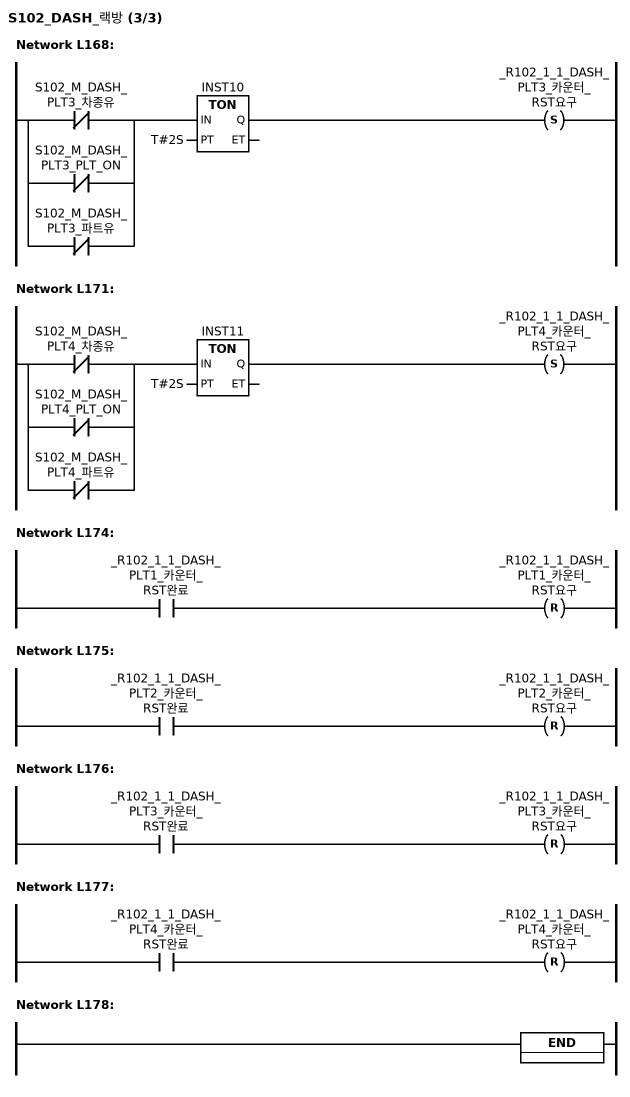
(* Rung L168 *)
INST10(IN := NOT S102_M_DASH_PLT3_차종유 OR NOT S102_M_DASH_PLT3_PLT_ON OR NOT S102_M_DASH_PLT3_파트유, PT := T#2S);
IF INST10.Q THEN _R102_1_1_DASH_PLT3_카운터_RST요구 := TRUE; END_IF;
(* Rung L171 *)
INST11(IN := NOT S102_M_DASH_PLT4_차종유 OR NOT S102_M_DASH_PLT4_PLT_ON OR NOT S102_M_DASH_PLT4_파트유, PT := T#2S);
IF INST11.Q THEN _R102_1_1_DASH_PLT4_카운터_RST요구 := TRUE; END_IF;
(* Rung L174 *)
IF _R102_1_1_DASH_PLT1_카운터_RST완료 THEN _R102_1_1_DASH_PLT1_카운터_RST요구 := FALSE; END_IF;
(* Rung L175 *)
IF _R102_1_1_DASH_PLT2_카운터_RST완료 THEN _R102_1_1_DASH_PLT2_카운터_RST요구 := FALSE; END_IF;
(* Rung L176 *)
IF _R102_1_1_DASH_PLT3_카운터_RST완료 THEN _R102_1_1_DASH_PLT3_카운터_RST요구 := FALSE; END_IF;
(* Rung L177 *)
IF _R102_1_1_DASH_PLT4_카운터_RST완료 THEN _R102_1_1_DASH_PLT4_카운터_RST요구 := FALSE; END_IF;
(* Rung L178 *)
END();
END_PROGRAM

PROGRAM S102_DASH_랙방_우선순위 (* task: 스캔 프로그램 *)
VAR_EXTERNAL
    S101_LH_M_APRON_PLT1_PLT_ON : BOOL; (* AT %MW1200.1 *)
    S101_LH_M_APRON_PLT1_로딩완료 : BOOL; (* AT %MW1200.10 *)
    S101_LH_M_APRON_PLT1_차종유 : BOOL; (* AT %MW1200.8 *)
    S101_LH_M_APRON_PLT1_파트유 : BOOL; (* AT %MW1200.3 *)
    S101_LH_M_APRON_PLT2_PLT_ON : BOOL; (* AT %MW1201.1 *)
    S101_LH_M_APRON_PLT2_로딩완료 : BOOL; (* AT %MW1201.10 *)
    S101_LH_M_APRON_PLT2_차종유 : BOOL; (* AT %MW1201.8 *)
    S101_LH_M_APRON_PLT2_파트유 : BOOL; (* AT %MW1201.3 *)
    S101_LH_M_APRON_PLT_PRIORITY1 : WORD; (* AT %MW1208 *)
    S101_LH_M_APRON_PLT_PRIORITY2 : WORD; (* AT %MW1209 *)
    S101_LH_M_APRON_PLT_PRIORITY3 : WORD; (* AT %MW1210 *)
    S101_LH_M_APRON_PLT_PRIORITY4 : WORD; (* AT %MW1211 *)
    S101_LH_M_APRON_PLT_PRIORITY5 : WORD; (* AT %MW1212 *)
    S101_LH_M_APRON_PLT_PRIORITY6 : WORD; (* AT %MW1213 *)
    S101_LH_M_APRON_PLT_PRIORITY7 : WORD; (* AT %MW1214 *)
    S101_LH_M_APRON_PLT_PRIORITY8 : WORD; (* AT %MW1215 *)
    S101_RH_M_APRON_PLT1_PLT_ON : BOOL; (* AT %MW1250.1 *)
    S101_RH_M_APRON_PLT1_로딩완료 : BOOL; (* AT %MW1250.10 *)
    S101_RH_M_APRON_PLT1_차종유 : BOOL; (* AT %MW1250.8 *)
    S101_RH_M_APRON_PLT1_파트유 : BOOL; (* AT %MW1250.3 *)
    S101_RH_M_APRON_PLT2_PLT_ON : BOOL; (* AT %MW1251.1 *)
    S101_RH_M_APRON_PLT2_로딩완료 : BOOL; (* AT %MW1251.10 *)
    S101_RH_M_APRON_PLT2_차종유 : BOOL; (* AT %MW1251.8 *)
    S101_RH_M_APRON_PLT2_파트유 : BOOL; (* AT %MW1251.3 *)
    S101_RH_M_APRON_PLT_PRIORITY1 : WORD; (* AT %MW1258 *)
    S101_RH_M_APRON_PLT_PRIORITY2 : WORD; (* AT %MW1259 *)
    S101_RH_M_APRON_PLT_PRIORITY3 : WORD; (* AT %MW1260 *)
    S101_RH_M_APRON_PLT_PRIORITY4 : WORD; (* AT %MW1261 *)
    S101_RH_M_APRON_PLT_PRIORITY5 : WORD; (* AT %MW1262 *)
    S101_RH_M_APRON_PLT_PRIORITY6 : WORD; (* AT %MW1263 *)
    S101_RH_M_APRON_PLT_PRIORITY7 : WORD; (* AT %MW1264 *)
    S101_RH_M_APRON_PLT_PRIORITY8 : WORD; (* AT %MW1265 *)
    S102_M_DASH_PLT1_PLT_ON : BOOL; (* AT %MW1700.1 *)
    S102_M_DASH_PLT1_로딩완료 : BOOL; (* AT %MW1700.10 *)
    S102_M_DASH_PLT1_차종유 : BOOL; (* AT %MW1700.8 *)
    S102_M_DASH_PLT1_파트유 : BOOL; (* AT %MW1700.3 *)
    S102_M_DASH_PLT2_PLT_ON : BOOL; (* AT %MW1701.1 *)
    S102_M_DASH_PLT2_로딩완료 : BOOL; (* AT %MW1701.10 *)
    S102_M_DASH_PLT2_차종유 : BOOL; (* AT %MW1701.8 *)
    S102_M_DASH_PLT2_파트유 : BOOL; (* AT %MW1701.3 *)
    S102_M_DASH_PLT3_PLT_ON : BOOL; (* AT %MW1702.1 *)
    S102_M_DASH_PLT3_로딩완료 : BOOL; (* AT %MW1702.10 *)
    S102_M_DASH_PLT3_차종유 : BOOL; (* AT %MW1702.8 *)
    S102_M_DASH_PLT3_파트유 : BOOL; (* AT %MW1702.3 *)
    S102_M_DASH_PLT4_PLT_ON : BOOL; (* AT %MW1703.1 *)
    S102_M_DASH_PLT4_로딩완료 : BOOL; (* AT %MW1703.10 *)
    S102_M_DASH_PLT4_차종유 : BOOL; (* AT %MW1703.8 *)
    S102_M_DASH_PLT4_파트유 : BOOL; (* AT %MW1703.3 *)
    S102_M_DASH_PLT_PRIORITY1 : WORD; (* AT %MW1708 *)
    S102_M_DASH_PLT_PRIORITY2 : WORD; (* AT %MW1709 *)
    S102_M_DASH_PLT_PRIORITY3 : WORD; (* AT %MW1710 *)
    S102_M_DASH_PLT_PRIORITY4 : WORD; (* AT %MW1711 *)
    S102_M_DASH_PLT_PRIORITY5 : WORD; (* AT %MW1712 *)
    S102_M_DASH_PLT_PRIORITY6 : WORD; (* AT %MW1713 *)
    S102_M_DASH_PLT_PRIORITY7 : WORD; (* AT %MW1714 *)
    S102_M_DASH_PLT_PRIORITY8 : WORD; (* AT %MW1715 *)
END_VAR
VAR
    _p1 : BOOL;
    _t2 : BOOL;
    _t3 : BOOL;
    _t4 : BOOL;
    _t5 : BOOL;
    _t6 : BOOL;
    _t7 : BOOL;
    _t8 : BOOL;
    _t9 : BOOL;
    _p10 : BOOL;
    _t11 : BOOL;
    _t12 : BOOL;
    _t13 : BOOL;
    _t14 : BOOL;
    _t15 : BOOL;
    _t16 : BOOL;
    _t17 : BOOL;
    _t18 : BOOL;
    _p19 : BOOL;
    _t20 : BOOL;
    _t21 : BOOL;
    _t22 : BOOL;
    _t23 : BOOL;
    _t24 : BOOL;
    _t25 : BOOL;
    _t26 : BOOL;
    _t27 : BOOL;
    _p28 : BOOL;
    _t29 : BOOL;
    _t30 : BOOL;
    _t31 : BOOL;
    _t32 : BOOL;
    _t33 : BOOL;
    _t34 : BOOL;
    _t35 : BOOL;
    _t36 : BOOL;
END_VAR
(* 랙방번호 우선순위버퍼 전송 *)
(* Rung L1: network not rendered *)
(* not connected or not rendered: S102_M_DASH_PLT1_로딩완료, S102_M_DASH_PLT1_PLT_ON, S102_M_DASH_PLT1_파트유, S102_M_DASH_PLT1_차종유, S102_M_DASH_PLT2_로딩완료, S102_M_DASH_PLT2_PLT_ON, S102_M_DASH_PLT2_파트유, S102_M_DASH_PLT2_차종유, S102_M_DASH_PLT3_로딩완료, S102_M_DASH_PLT3_PLT_ON, S102_M_DASH_PLT3_파트유, S102_M_DASH_PLT3_차종유, S102_M_DASH_PLT4_로딩완료, S102_M_DASH_PLT4_PLT_ON, S102_M_DASH_PLT4_파트유, S102_M_DASH_PLT4_차종유, S102_M_DASH_PLT_PRIORITY8, 0, S102_M_DASH_PLT_PRIORITY8, 2, S102_M_DASH_PLT_PRIORITY8, 3, S102_M_DASH_PLT_PRIORITY8, 4, S102_M_DASH_PLT_PRIORITY8 *)
(* 우선순위8->우선순위7 *)
(* Rung L15: network not rendered *)
(* not connected or not rendered: S102_M_DASH_PLT_PRIORITY8, 0, S102_M_DASH_PLT_PRIORITY7, 0, S102_M_DASH_PLT_PRIORITY8, S102_M_DASH_PLT_PRIORITY7, 0, S102_M_DASH_PLT_PRIORITY8 *)
(* 우선순위7->우선순위6 *)
(* Rung L24: network not rendered *)
(* not connected or not rendered: S102_M_DASH_PLT_PRIORITY7, 0, S102_M_DASH_PLT_PRIORITY6, 0, S102_M_DASH_PLT_PRIORITY7, S102_M_DASH_PLT_PRIORITY6, 0, S102_M_DASH_PLT_PRIORITY7 *)
(* 우선순위6->우선순위5 *)
(* Rung L33: network not rendered *)
(* not connected or not rendered: S102_M_DASH_PLT_PRIORITY6, 0, S102_M_DASH_PLT_PRIORITY5, 0, S102_M_DASH_PLT_PRIORITY6, S102_M_DASH_PLT_PRIORITY5, 0, S102_M_DASH_PLT_PRIORITY6 *)
(* 우선순위5->우선순위4 *)
(* Rung L42: network not rendered *)
(* not connected or not rendered: S102_M_DASH_PLT_PRIORITY5, 0, S102_M_DASH_PLT_PRIORITY4, 0, S102_M_DASH_PLT_PRIORITY5, S102_M_DASH_PLT_PRIORITY4, 0, S102_M_DASH_PLT_PRIORITY5 *)
(* 우선순위4->우선순위3 *)
(* Rung L51: network not rendered *)
(* not connected or not rendered: S102_M_DASH_PLT_PRIORITY4, 0, S102_M_DASH_PLT_PRIORITY3, 0, S102_M_DASH_PLT_PRIORITY4, S102_M_DASH_PLT_PRIORITY3, 0, S102_M_DASH_PLT_PRIORITY4 *)
(* 우선순위3->우선순위2 *)
(* Rung L60: network not rendered *)
(* not connected or not rendered: S102_M_DASH_PLT_PRIORITY3, S102_M_DASH_PLT_PRIORITY2, S102_M_DASH_PLT_PRIORITY3, S102_M_DASH_PLT_PRIORITY2, S102_M_DASH_PLT_PRIORITY3 *)
(* 우선순위2->우선순위1 *)
(* Rung L69: network not rendered *)
(* not connected or not rendered: S102_M_DASH_PLT_PRIORITY2, 0, S102_M_DASH_PLT_PRIORITY1, 0, S102_M_DASH_PLT_PRIORITY2, S102_M_DASH_PLT_PRIORITY1, 0, S102_M_DASH_PLT_PRIORITY2 *)

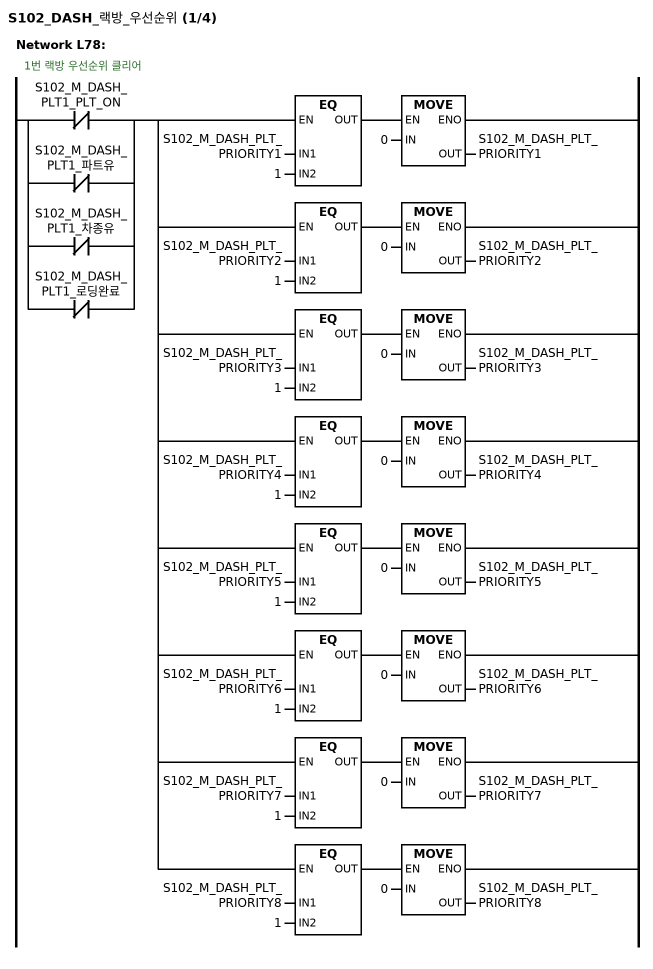
(* 1번 랙방 우선순위 클리어 *)
(* Rung L78 *)
_p1 := NOT S102_M_DASH_PLT1_PLT_ON OR NOT S102_M_DASH_PLT1_파트유 OR NOT S102_M_DASH_PLT1_차종유 OR NOT S102_M_DASH_PLT1_로딩완료;
IF _p1 THEN _t2 := S102_M_DASH_PLT_PRIORITY1 = 1; END_IF;
IF _t2 THEN S102_M_DASH_PLT_PRIORITY1 := 0; END_IF;
IF _p1 THEN _t3 := S102_M_DASH_PLT_PRIORITY2 = 1; END_IF;
IF _t3 THEN S102_M_DASH_PLT_PRIORITY2 := 0; END_IF;
IF _p1 THEN _t4 := S102_M_DASH_PLT_PRIORITY3 = 1; END_IF;
IF _t4 THEN S102_M_DASH_PLT_PRIORITY3 := 0; END_IF;
IF _p1 THEN _t5 := S102_M_DASH_PLT_PRIORITY4 = 1; END_IF;
IF _t5 THEN S102_M_DASH_PLT_PRIORITY4 := 0; END_IF;
IF _p1 THEN _t6 := S102_M_DASH_PLT_PRIORITY5 = 1; END_IF;
IF _t6 THEN S102_M_DASH_PLT_PRIORITY5 := 0; END_IF;
IF _p1 THEN _t7 := S102_M_DASH_PLT_PRIORITY6 = 1; END_IF;
IF _t7 THEN S102_M_DASH_PLT_PRIORITY6 := 0; END_IF;
IF _p1 THEN _t8 := S102_M_DASH_PLT_PRIORITY7 = 1; END_IF;
IF _t8 THEN S102_M_DASH_PLT_PRIORITY7 := 0; END_IF;
IF _p1 THEN _t9 := S102_M_DASH_PLT_PRIORITY8 = 1; END_IF;
IF _t9 THEN S102_M_DASH_PLT_PRIORITY8 := 0; END_IF;

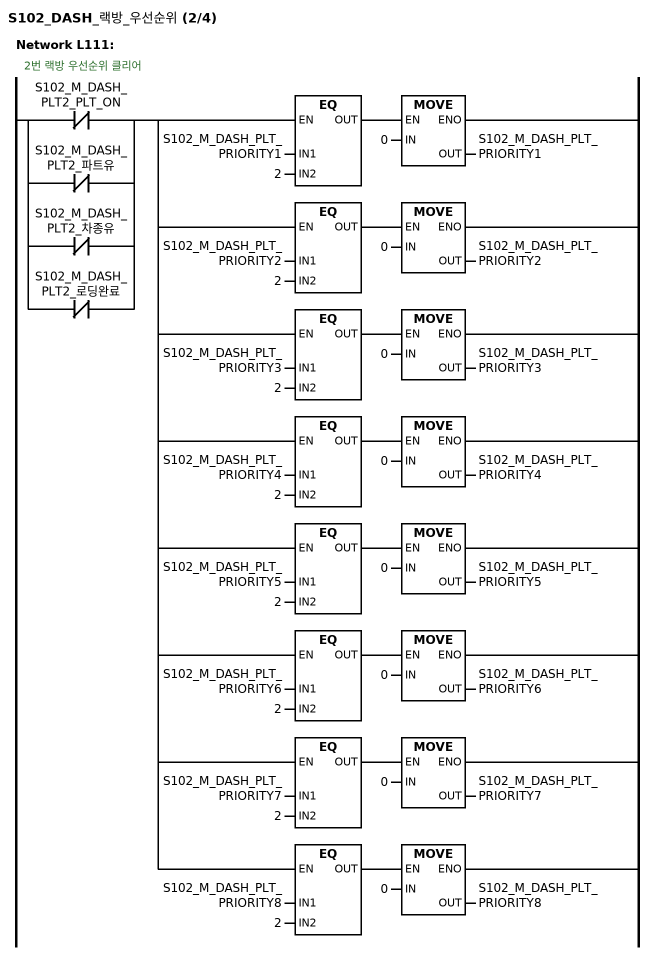
(* 2번 랙방 우선순위 클리어 *)
(* Rung L111 *)
_p10 := NOT S102_M_DASH_PLT2_PLT_ON OR NOT S102_M_DASH_PLT2_파트유 OR NOT S102_M_DASH_PLT2_차종유 OR NOT S102_M_DASH_PLT2_로딩완료;
IF _p10 THEN _t11 := S102_M_DASH_PLT_PRIORITY1 = 2; END_IF;
IF _t11 THEN S102_M_DASH_PLT_PRIORITY1 := 0; END_IF;
IF _p10 THEN _t12 := S102_M_DASH_PLT_PRIORITY2 = 2; END_IF;
IF _t12 THEN S102_M_DASH_PLT_PRIORITY2 := 0; END_IF;
IF _p10 THEN _t13 := S102_M_DASH_PLT_PRIORITY3 = 2; END_IF;
IF _t13 THEN S102_M_DASH_PLT_PRIORITY3 := 0; END_IF;
IF _p10 THEN _t14 := S102_M_DASH_PLT_PRIORITY4 = 2; END_IF;
IF _t14 THEN S102_M_DASH_PLT_PRIORITY4 := 0; END_IF;
IF _p10 THEN _t15 := S102_M_DASH_PLT_PRIORITY5 = 2; END_IF;
IF _t15 THEN S102_M_DASH_PLT_PRIORITY5 := 0; END_IF;
IF _p10 THEN _t16 := S102_M_DASH_PLT_PRIORITY6 = 2; END_IF;
IF _t16 THEN S102_M_DASH_PLT_PRIORITY6 := 0; END_IF;
IF _p10 THEN _t17 := S102_M_DASH_PLT_PRIORITY7 = 2; END_IF;
IF _t17 THEN S102_M_DASH_PLT_PRIORITY7 := 0; END_IF;
IF _p10 THEN _t18 := S102_M_DASH_PLT_PRIORITY8 = 2; END_IF;
IF _t18 THEN S102_M_DASH_PLT_PRIORITY8 := 0; END_IF;

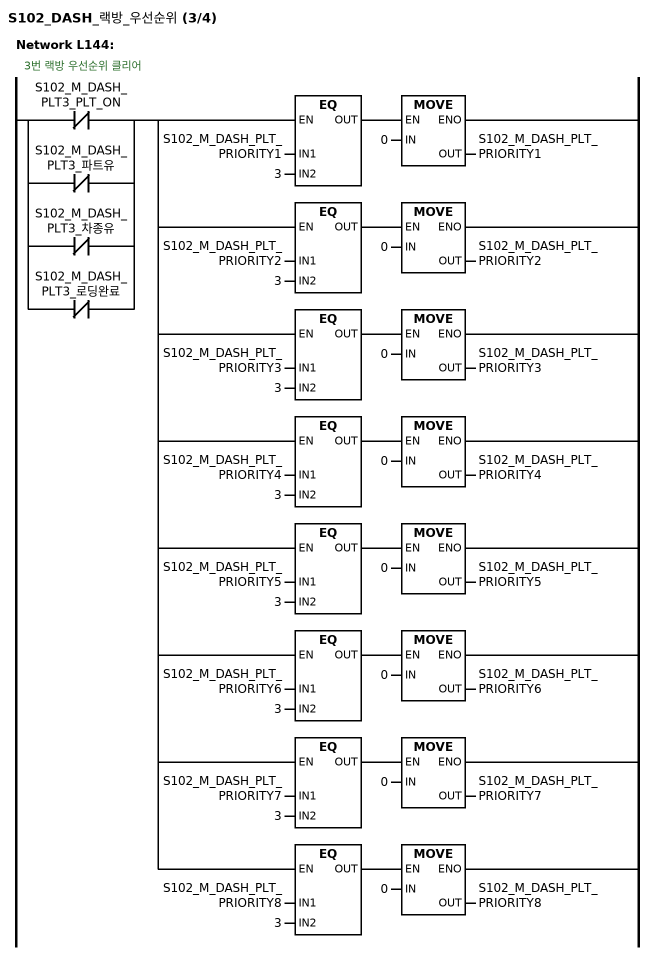
(* 3번 랙방 우선순위 클리어 *)
(* Rung L144 *)
_p19 := NOT S102_M_DASH_PLT3_PLT_ON OR NOT S102_M_DASH_PLT3_파트유 OR NOT S102_M_DASH_PLT3_차종유 OR NOT S102_M_DASH_PLT3_로딩완료;
IF _p19 THEN _t20 := S102_M_DASH_PLT_PRIORITY1 = 3; END_IF;
IF _t20 THEN S102_M_DASH_PLT_PRIORITY1 := 0; END_IF;
IF _p19 THEN _t21 := S102_M_DASH_PLT_PRIORITY2 = 3; END_IF;
IF _t21 THEN S102_M_DASH_PLT_PRIORITY2 := 0; END_IF;
IF _p19 THEN _t22 := S102_M_DASH_PLT_PRIORITY3 = 3; END_IF;
IF _t22 THEN S102_M_DASH_PLT_PRIORITY3 := 0; END_IF;
IF _p19 THEN _t23 := S102_M_DASH_PLT_PRIORITY4 = 3; END_IF;
IF _t23 THEN S102_M_DASH_PLT_PRIORITY4 := 0; END_IF;
IF _p19 THEN _t24 := S102_M_DASH_PLT_PRIORITY5 = 3; END_IF;
IF _t24 THEN S102_M_DASH_PLT_PRIORITY5 := 0; END_IF;
IF _p19 THEN _t25 := S102_M_DASH_PLT_PRIORITY6 = 3; END_IF;
IF _t25 THEN S102_M_DASH_PLT_PRIORITY6 := 0; END_IF;
IF _p19 THEN _t26 := S102_M_DASH_PLT_PRIORITY7 = 3; END_IF;
IF _t26 THEN S102_M_DASH_PLT_PRIORITY7 := 0; END_IF;
IF _p19 THEN _t27 := S102_M_DASH_PLT_PRIORITY8 = 3; END_IF;
IF _t27 THEN S102_M_DASH_PLT_PRIORITY8 := 0; END_IF;

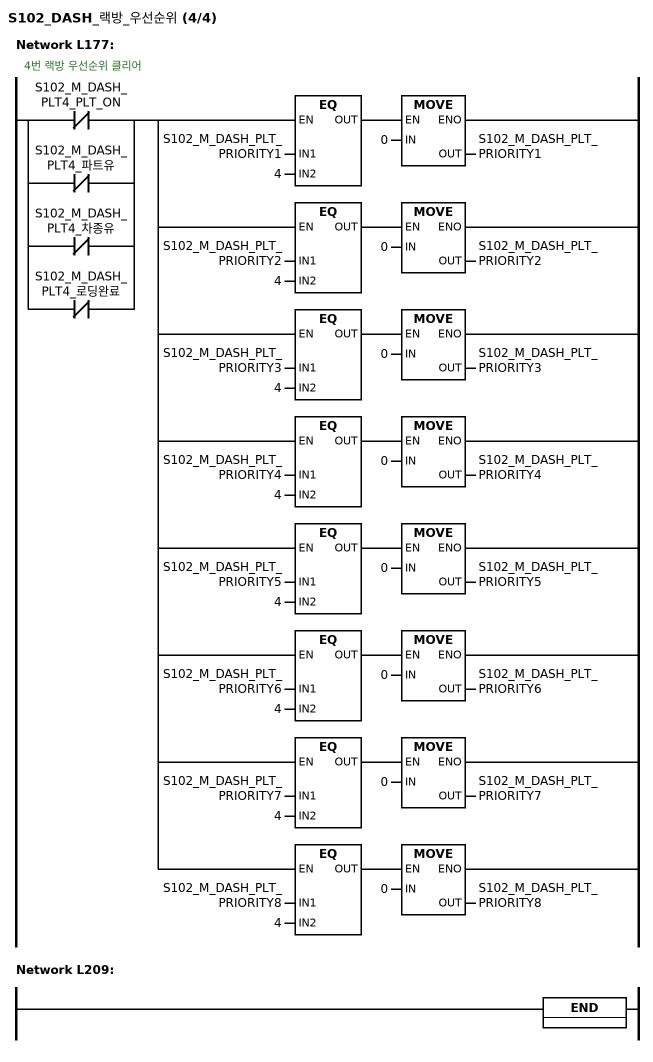
(* 4번 랙방 우선순위 클리어 *)
(* Rung L177 *)
_p28 := NOT S102_M_DASH_PLT4_PLT_ON OR NOT S102_M_DASH_PLT4_파트유 OR NOT S102_M_DASH_PLT4_차종유 OR NOT S102_M_DASH_PLT4_로딩완료;
IF _p28 THEN _t29 := S102_M_DASH_PLT_PRIORITY1 = 4; END_IF;
IF _t29 THEN S102_M_DASH_PLT_PRIORITY1 := 0; END_IF;
IF _p28 THEN _t30 := S102_M_DASH_PLT_PRIORITY2 = 4; END_IF;
IF _t30 THEN S102_M_DASH_PLT_PRIORITY2 := 0; END_IF;
IF _p28 THEN _t31 := S102_M_DASH_PLT_PRIORITY3 = 4; END_IF;
IF _t31 THEN S102_M_DASH_PLT_PRIORITY3 := 0; END_IF;
IF _p28 THEN _t32 := S102_M_DASH_PLT_PRIORITY4 = 4; END_IF;
IF _t32 THEN S102_M_DASH_PLT_PRIORITY4 := 0; END_IF;
IF _p28 THEN _t33 := S102_M_DASH_PLT_PRIORITY5 = 4; END_IF;
IF _t33 THEN S102_M_DASH_PLT_PRIORITY5 := 0; END_IF;
IF _p28 THEN _t34 := S102_M_DASH_PLT_PRIORITY6 = 4; END_IF;
IF _t34 THEN S102_M_DASH_PLT_PRIORITY6 := 0; END_IF;
IF _p28 THEN _t35 := S102_M_DASH_PLT_PRIORITY7 = 4; END_IF;
IF _t35 THEN S102_M_DASH_PLT_PRIORITY7 := 0; END_IF;
IF _p28 THEN _t36 := S102_M_DASH_PLT_PRIORITY8 = 4; END_IF;
IF _t36 THEN S102_M_DASH_PLT_PRIORITY8 := 0; END_IF;
(* Rung L209 *)
END();
END_PROGRAM

PROGRAM S102_로보트 (* task: 스캔 프로그램 *)
VAR_EXTERNAL
    AWAYS_OFF : BOOL; (* AT %MW3.0 *)
    AWAYS_ON : BOOL; (* AT %MW3.1 *)
    MCP_M_부저_정지 : BOOL; (* AT %MW350.5 *)
    MCP_M_비상정지 : BOOL; (* AT %MW350.7 *)
    MCP_PBL_운전준비_ON : BOOL; (* AT %MW87630.0 *) (* 입력 접점 00 *)
    R101_1_1_M_I_RB_간섭무_2 : BOOL; (* AT %MW20042.1 *)
    R101_1_M_I_RB_간섭무_2 : BOOL; (* AT %MW20072.1 *)
    R101_2_M_I_RB_간섭무_2 : BOOL; (* AT %MW20062.1 *)
    R101_3_M_I_RB_간섭무_2 : BOOL; (* AT %MW20052.1 *)
    R102_1_1_I_RB_INPUT : ARRAY[0..3] OF WORD; (* AT %MW84090 *)
    R102_1_1_M_I_RB_1차_작업완료 : BOOL; (* AT %MW20091.2 *)
    R102_1_1_M_I_RB_2차_작업완료 : BOOL; (* AT %MW20091.3 *)
    R102_1_1_M_I_RB_3차_작업완료 : BOOL; (* AT %MW20091.4 *)
    R102_1_1_M_I_RB_4차_작업완료 : BOOL; (* AT %MW20091.5 *)
    R102_1_1_M_I_RB_5차_작업완료 : BOOL; (* AT %MW20091.6 *)
    R102_1_1_M_I_RB_6차_작업완료 : BOOL; (* AT %MW20091.7 *)
    R102_1_1_M_I_RB_7차_작업완료 : BOOL; (* AT %MW20091.8 *)
    R102_1_1_M_I_RB_PAUSE_보조 : BOOL; (* AT %MW20090.5 *)
    R102_1_1_M_I_RB_PLC_RUN_CHK_이상 : BOOL; (* AT %MW20090.7 *)
    R102_1_1_M_I_RB_간섭무_1 : BOOL; (* AT %MW20092.0 *)
    R102_1_1_M_I_RB_간섭무_10 : BOOL; (* AT %MW20092.9 *)
    R102_1_1_M_I_RB_간섭무_11 : BOOL; (* AT %MW20092.10 *)
    R102_1_1_M_I_RB_간섭무_12 : BOOL; (* AT %MW20092.11 *)
    R102_1_1_M_I_RB_간섭무_2 : BOOL; (* AT %MW20092.1 *)
    R102_1_1_M_I_RB_간섭무_3 : BOOL; (* AT %MW20092.2 *)
    R102_1_1_M_I_RB_간섭무_4 : BOOL; (* AT %MW20092.3 *)
    R102_1_1_M_I_RB_간섭무_5 : BOOL; (* AT %MW20092.4 *)
    R102_1_1_M_I_RB_간섭무_6 : BOOL; (* AT %MW20092.5 *)
    R102_1_1_M_I_RB_간섭무_7 : BOOL; (* AT %MW20092.6 *)
    R102_1_1_M_I_RB_간섭무_8 : BOOL; (* AT %MW20092.7 *)
    R102_1_1_M_I_RB_간섭무_9 : BOOL; (* AT %MW20092.8 *)
    R102_1_1_M_I_RB_비상정지 : BOOL; (* AT %MW20090.4 *)
    R102_1_1_M_I_RB_운전준비 : BOOL; (* AT %MW20090.0 *)
    R102_1_1_M_I_RB_원위치 : BOOL; (* AT %MW20090.3 *)
    R102_1_1_M_I_RB_이상 : BOOL; (* AT %MW20090.2 *)
    R102_1_1_M_I_RB_자동 : BOOL; (* AT %MW20090.1 *)
    R102_1_1_M_I_RB_최종작업완료 : BOOL; (* AT %MW20091.0 *)
    R102_1_1_M_I_RB_프로그램_이상 : BOOL; (* AT %MW20090.6 *)
    R102_1_1_M_O_RB_1_CYCLE_SET : BOOL; (* AT %MW21090.3 *)
    R102_1_1_M_O_RB_1차_작업완료_리셋 : BOOL; (* AT %MW21092.0 *)
    R102_1_1_M_O_RB_2차_작업완료_리셋 : BOOL; (* AT %MW21092.1 *)
    R102_1_1_M_O_RB_2차_진입OK : BOOL; (* AT %MW21091.8 *)
    R102_1_1_M_O_RB_3차_작업완료_리셋 : BOOL; (* AT %MW21092.2 *)
    R102_1_1_M_O_RB_3차_진입OK : BOOL; (* AT %MW21091.9 *)
    R102_1_1_M_O_RB_4차_작업완료_리셋 : BOOL; (* AT %MW21092.3 *)
    R102_1_1_M_O_RB_4차_진입OK : BOOL; (* AT %MW21091.10 *)
    R102_1_1_M_O_RB_5차_작업완료_리셋 : BOOL; (* AT %MW21092.4 *)
    R102_1_1_M_O_RB_5차_진입OK : BOOL; (* AT %MW21091.11 *)
    R102_1_1_M_O_RB_6차_작업완료_리셋 : BOOL; (* AT %MW21092.5 *)
    R102_1_1_M_O_RB_6차_진입OK : BOOL; (* AT %MW21091.12 *)
    R102_1_1_M_O_RB_7차_작업완료_리셋 : BOOL; (* AT %MW21092.6 *)
    R102_1_1_M_O_RB_7차_진입OK : BOOL; (* AT %MW21091.13 *)
    R102_1_1_M_O_RB_ATD_OK : BOOL; (* AT %MW21090.6 *)
    R102_1_1_M_O_RB_PLT_10_진입OK : BOOL; (* AT %MW21093.10 *)
    R102_1_1_M_O_RB_PLT_11_진입OK : BOOL; (* AT %MW21093.11 *)
    R102_1_1_M_O_RB_PLT_12_진입OK : BOOL; (* AT %MW21093.12 *)
    R102_1_1_M_O_RB_PLT_1_진입OK : BOOL; (* AT %MW21093.1 *)
    R102_1_1_M_O_RB_PLT_2_진입OK : BOOL; (* AT %MW21093.2 *)
    R102_1_1_M_O_RB_PLT_3_진입OK : BOOL; (* AT %MW21093.3 *)
    R102_1_1_M_O_RB_PLT_4_진입OK : BOOL; (* AT %MW21093.4 *)
    R102_1_1_M_O_RB_PLT_5_진입OK : BOOL; (* AT %MW21093.5 *)
    R102_1_1_M_O_RB_PLT_6_진입OK : BOOL; (* AT %MW21093.6 *)
    R102_1_1_M_O_RB_PLT_7_진입OK : BOOL; (* AT %MW21093.7 *)
    R102_1_1_M_O_RB_PLT_8_진입OK : BOOL; (* AT %MW21093.8 *)
    R102_1_1_M_O_RB_PLT_9_진입OK : BOOL; (* AT %MW21093.9 *)
    R102_1_1_M_O_RB_PLT_카운터리셋_보조 : BOOL; (* AT %MW21090.10 *)
    R102_1_1_M_O_RB_RESTART_OK : BOOL; (* AT %MW21090.2 *)
    R102_1_1_M_O_RB_START_OK : BOOL; (* AT %MW21090.0 *)
    R102_1_1_M_O_RB_TEST_MODE_5000회 : BOOL; (* AT %MW21090.12 *)
    R102_1_1_M_O_RB_TIP_교체_시작 : BOOL; (* AT %MW21090.7 *)
    R102_1_1_M_O_RB_TIP_교체_완료 : BOOL; (* AT %MW21090.8 *)
    R102_1_1_M_O_RB_VIP_MODE : BOOL; (* AT %MW21090.11 *)
    R102_1_1_M_O_RB_냉각수_차단_요청 : BOOL; (* AT %MW21090.9 *)
    R102_1_1_M_O_RB_진입OK_AX차종 : BOOL; (* AT %MW21091.0 *)
    R102_1_1_M_O_RB_진입OK_B차종 : BOOL; (* AT %MW21091.1 *)
    R102_1_1_M_O_RB_진입OK_C차종 : BOOL; (* AT %MW21091.2 *)
    R102_1_1_M_O_RB_진입OK_D차종 : BOOL; (* AT %MW21091.3 *)
    R102_1_1_M_O_RB_진입OK_E차종 : BOOL; (* AT %MW21091.4 *)
    R102_1_1_M_O_RB_진입OK_F차종 : BOOL; (* AT %MW21091.5 *)
    R102_1_1_M_O_RB_진입OK_G차종 : BOOL; (* AT %MW21091.6 *)
    R102_1_1_M_O_RB_진입OK_H차종 : BOOL; (* AT %MW21091.7 *)
    R102_1_1_M_O_RB_최종_작업완료_리셋 : BOOL; (* AT %MW21090.5 *)
    R102_1_1_M_O_RB_프로그램_OK : BOOL; (* AT %MW21090.1 *)
    R102_1_1_M_RB_PROG_NO : WORD; (* AT %MW20094 *)
    R102_1_1_M_STN_차종_NONE : BOOL; (* AT %MW1502.3 *)
    R102_1_1_M_STN_차종_ON : BOOL; (* AT %MW1502.2 *)
    R102_1_1_M_차종1_AX : BOOL; (* AT %MW10041.0 *) (* R102_1_1_M_차종1_AX *)
    R102_1_1_O_RB_OUTPUT : ARRAY[0..3] OF WORD; (* AT %MW94090 *)
    R102_1_I_RB_INPUT : ARRAY[0..3] OF WORD; (* AT %MW84080 *)
    R102_1_M_I_RB_1차_작업완료 : BOOL; (* AT %MW20081.2 *)
    R102_1_M_I_RB_2차_작업완료 : BOOL; (* AT %MW20081.3 *)
    R102_1_M_I_RB_3차_작업완료 : BOOL; (* AT %MW20081.4 *)
    R102_1_M_I_RB_4차_작업완료 : BOOL; (* AT %MW20081.5 *)
    R102_1_M_I_RB_5차_작업완료 : BOOL; (* AT %MW20081.6 *)
    R102_1_M_I_RB_6차_작업완료 : BOOL; (* AT %MW20081.7 *)
    R102_1_M_I_RB_7차_작업완료 : BOOL; (* AT %MW20081.8 *)
    R102_1_M_I_RB_PAUSE_보조 : BOOL; (* AT %MW20080.5 *)
    R102_1_M_I_RB_PLC_RUN_CHK_이상 : BOOL; (* AT %MW20080.7 *)
    R102_1_M_I_RB_간섭무_1 : BOOL; (* AT %MW20082.0 *)
    R102_1_M_I_RB_간섭무_10 : BOOL; (* AT %MW20082.9 *)
    R102_1_M_I_RB_간섭무_11 : BOOL; (* AT %MW20082.10 *)
    R102_1_M_I_RB_간섭무_12 : BOOL; (* AT %MW20082.11 *)
    R102_1_M_I_RB_간섭무_2 : BOOL; (* AT %MW20082.1 *)
    R102_1_M_I_RB_간섭무_3 : BOOL; (* AT %MW20082.2 *)
    R102_1_M_I_RB_간섭무_4 : BOOL; (* AT %MW20082.3 *)
    R102_1_M_I_RB_간섭무_5 : BOOL; (* AT %MW20082.4 *)
    R102_1_M_I_RB_간섭무_6 : BOOL; (* AT %MW20082.5 *)
    R102_1_M_I_RB_간섭무_7 : BOOL; (* AT %MW20082.6 *)
    R102_1_M_I_RB_간섭무_8 : BOOL; (* AT %MW20082.7 *)
    R102_1_M_I_RB_간섭무_9 : BOOL; (* AT %MW20082.8 *)
    R102_1_M_I_RB_비상정지 : BOOL; (* AT %MW20080.4 *)
    R102_1_M_I_RB_운전준비 : BOOL; (* AT %MW20080.0 *)
    R102_1_M_I_RB_원위치 : BOOL; (* AT %MW20080.3 *)
    R102_1_M_I_RB_이상 : BOOL; (* AT %MW20080.2 *)
    R102_1_M_I_RB_자동 : BOOL; (* AT %MW20080.1 *)
    R102_1_M_I_RB_최종작업완료 : BOOL; (* AT %MW20081.0 *)
    R102_1_M_I_RB_프로그램_이상 : BOOL; (* AT %MW20080.6 *)
    R102_1_M_O_RB_1_CYCLE_SET : BOOL; (* AT %MW21080.3 *)
    R102_1_M_O_RB_1차_작업완료_리셋 : BOOL; (* AT %MW21082.0 *)
    R102_1_M_O_RB_2차_작업완료_리셋 : BOOL; (* AT %MW21082.1 *)
    R102_1_M_O_RB_2차_진입OK : BOOL; (* AT %MW21081.8 *)
    R102_1_M_O_RB_3차_작업완료_리셋 : BOOL; (* AT %MW21082.2 *)
    R102_1_M_O_RB_3차_진입OK : BOOL; (* AT %MW21081.9 *)
    R102_1_M_O_RB_4차_작업완료_리셋 : BOOL; (* AT %MW21082.3 *)
    R102_1_M_O_RB_4차_진입OK : BOOL; (* AT %MW21081.10 *)
    R102_1_M_O_RB_5차_작업완료_리셋 : BOOL; (* AT %MW21082.4 *)
    R102_1_M_O_RB_5차_진입OK : BOOL; (* AT %MW21081.11 *)
    R102_1_M_O_RB_6차_작업완료_리셋 : BOOL; (* AT %MW21082.5 *)
    R102_1_M_O_RB_6차_진입OK : BOOL; (* AT %MW21081.12 *)
    R102_1_M_O_RB_7차_작업완료_리셋 : BOOL; (* AT %MW21082.6 *)
    R102_1_M_O_RB_7차_진입OK : BOOL; (* AT %MW21081.13 *)
    R102_1_M_O_RB_ATD_OK : BOOL; (* AT %MW21080.6 *)
    R102_1_M_O_RB_PLT_10_진입OK : BOOL; (* AT %MW21083.10 *)
    R102_1_M_O_RB_PLT_11_진입OK : BOOL; (* AT %MW21083.11 *)
    R102_1_M_O_RB_PLT_12_진입OK : BOOL; (* AT %MW21083.12 *)
    R102_1_M_O_RB_PLT_1_진입OK : BOOL; (* AT %MW21083.1 *)
    R102_1_M_O_RB_PLT_2_진입OK : BOOL; (* AT %MW21083.2 *)
    R102_1_M_O_RB_PLT_3_진입OK : BOOL; (* AT %MW21083.3 *)
    R102_1_M_O_RB_PLT_4_진입OK : BOOL; (* AT %MW21083.4 *)
    R102_1_M_O_RB_PLT_5_진입OK : BOOL; (* AT %MW21083.5 *)
    R102_1_M_O_RB_PLT_6_진입OK : BOOL; (* AT %MW21083.6 *)
    R102_1_M_O_RB_PLT_7_진입OK : BOOL; (* AT %MW21083.7 *)
    R102_1_M_O_RB_PLT_8_진입OK : BOOL; (* AT %MW21083.8 *)
    R102_1_M_O_RB_PLT_9_진입OK : BOOL; (* AT %MW21083.9 *)
    R102_1_M_O_RB_PLT_카운터리셋_보조 : BOOL; (* AT %MW21080.10 *)
    R102_1_M_O_RB_RESTART_OK : BOOL; (* AT %MW21080.2 *)
    R102_1_M_O_RB_START_OK : BOOL; (* AT %MW21080.0 *)
    R102_1_M_O_RB_TEST_MODE_5000회 : BOOL; (* AT %MW21080.12 *)
    R102_1_M_O_RB_TIP_교체_시작 : BOOL; (* AT %MW21080.7 *)
    R102_1_M_O_RB_TIP_교체_완료 : BOOL; (* AT %MW21080.8 *)
    R102_1_M_O_RB_VIP_MODE : BOOL; (* AT %MW21080.11 *)
    R102_1_M_O_RB_냉각수_차단_요청 : BOOL; (* AT %MW21080.9 *)
    R102_1_M_O_RB_진입OK_AX차종 : BOOL; (* AT %MW21081.0 *)
    R102_1_M_O_RB_진입OK_B차종 : BOOL; (* AT %MW21081.1 *)
    R102_1_M_O_RB_진입OK_C차종 : BOOL; (* AT %MW21081.2 *)
    R102_1_M_O_RB_진입OK_D차종 : BOOL; (* AT %MW21081.3 *)
    R102_1_M_O_RB_진입OK_E차종 : BOOL; (* AT %MW21081.4 *)
    R102_1_M_O_RB_진입OK_F차종 : BOOL; (* AT %MW21081.5 *)
    R102_1_M_O_RB_진입OK_G차종 : BOOL; (* AT %MW21081.6 *)
    R102_1_M_O_RB_진입OK_H차종 : BOOL; (* AT %MW21081.7 *)
    R102_1_M_O_RB_최종_작업완료_리셋 : BOOL; (* AT %MW21080.5 *)
    R102_1_M_O_RB_프로그램_OK : BOOL; (* AT %MW21080.1 *)
    R102_1_M_RB_PROG_NO : WORD; (* AT %MW20084 *)
    R102_1_M_STN_차종_ON : BOOL; (* AT %MW1502.4 *)
    R102_1_M_차종1_AX : BOOL; (* AT %MW10081.0 *) (* R102_1_M_차종1_AX *)
    R102_1_O_RB_OUTPUT : ARRAY[0..3] OF WORD; (* AT %MW94080 *)
    R103_1_M_I_RB_간섭무_2 : BOOL; (* AT %MW20102.1 *)
    S101_M_STN_DASH_로딩완료 : BOOL; (* AT %MW1001.12 *)
    S101_M_STN_LH_로딩완료 : BOOL; (* AT %MW1001.10 *)
    S101_M_STN_RH_로딩완료 : BOOL; (* AT %MW1001.11 *)
    S101_M_STN_차종_ON : BOOL; (* AT %MW1002.0 *)
    S101_M_공정_APRON_제품감지_ON : BOOL; (* AT %MW1001.3 *)
    S101_M_공정_DASH_제품감지_OFF : BOOL; (* AT %MW1001.6 *)
    S101_M_공정_DASH_제품감지_ON : BOOL; (* AT %MW1001.5 *)
    S101_M_공정_간섭무 : BOOL; (* AT %MW1004.1 *)
    S101_M_자동_운전중 : BOOL; (* AT %MW1000.4 *)
    S101_M_작업_완료 : BOOL; (* AT %MW1001.0 *)
    S101_M_차종1_AX : BOOL; (* AT %MW10021.0 *) (* S101_M_차종1_AX *)
    S102_M_DASH_PLT1_FAULT : BOOL; (* AT %MW1700.6 *)
    S102_M_DASH_PLT1_MATCH_OK : BOOL; (* AT %MW1700.5 *)
    S102_M_DASH_PLT1_PROG_OK : BOOL; (* AT %MW1700.0 *)
    S102_M_DASH_PLT1_차종코드 : WORD; (* AT %MW1716 *)
    S102_M_DASH_PLT2_FAULT : BOOL; (* AT %MW1701.6 *)
    S102_M_DASH_PLT2_MATCH_OK : BOOL; (* AT %MW1701.5 *)
    S102_M_DASH_PLT2_PROG_OK : BOOL; (* AT %MW1701.0 *)
    S102_M_DASH_PLT2_차종코드 : WORD; (* AT %MW1717 *)
    S102_M_DASH_PLT3_FAULT : BOOL; (* AT %MW1702.6 *)
    S102_M_DASH_PLT3_MATCH_OK : BOOL; (* AT %MW1702.5 *)
    S102_M_DASH_PLT3_PROG_OK : BOOL; (* AT %MW1702.0 *)
    S102_M_DASH_PLT3_차종코드 : WORD; (* AT %MW1718 *)
    S102_M_DASH_PLT4_FAULT : BOOL; (* AT %MW1703.6 *)
    S102_M_DASH_PLT4_MATCH_OK : BOOL; (* AT %MW1703.5 *)
    S102_M_DASH_PLT4_PROG_OK : BOOL; (* AT %MW1703.0 *)
    S102_M_DASH_PLT4_차종코드 : WORD; (* AT %MW1719 *)
    S102_M_DASH_PLT_PRIORITY1 : WORD; (* AT %MW1708 *)
    S102_M_STN_차종_NONE : BOOL; (* AT %MW1502.1 *)
    S102_M_STN_차종_ON : BOOL; (* AT %MW1502.0 *)
    S102_M_공정_간섭무 : BOOL; (* AT %MW1504.1 *)
    S102_M_공정_사양감지_OK : BOOL; (* AT %MW1501.5 *)
    S102_M_공정_제품감지_OFF : BOOL; (* AT %MW1501.4 *)
    S102_M_공정_제품감지_ON : BOOL; (* AT %MW1501.3 *)
    S102_M_자동_START : BOOL; (* AT %MW1500.5 *)
    S102_M_자동_운전중 : BOOL; (* AT %MW1500.4 *)
    S102_M_작업_완료 : BOOL; (* AT %MW1501.0 *)
    S102_M_차종1_AX : BOOL; (* AT %MW10061.0 *) (* S102_M_차종1_AX *)
    S102_M_총괄_이상 : BOOL; (* AT %MW1509.0 *)
    S103_M_FRT_안착OK_POS : BOOL; (* AT %MW2004.8 *)
    S103_M_STN_차종_NONE : BOOL; (* AT %MW2002.1 *)
    S103_M_STN_차종_ON : BOOL; (* AT %MW2002.0 *)
    S103_M_공정_제품감지_OFF : BOOL; (* AT %MW2001.4 *)
    S103_M_자동_운전중 : BOOL; (* AT %MW2000.4 *)
    S103_M_작업_완료 : BOOL; (* AT %MW2001.0 *)
    로보트제외 : BOOL;
    전체_M_GATE_CYCLE_정지 : BOOL; (* AT %MW308.0 *) (* 전체 M GATE CYCLE STOP *)
    전체_M_GATE_비상정지_정상 : BOOL; (* AT %MW308.4 *)
    전체_M_운전준비_보조 : BOOL; (* AT %MW308.5 *)
    전체_M_이상_리셋 : BOOL; (* AT %MW308.2 *) (* 전체 M 이상 리셋 *)
    전체_공정_M_총괄_비상정지_정상 : BOOL; (* AT %MW304.1 *) (* 전체 공정 M 총괄 비상정지 정상 *)
END_VAR
VAR
    INST1 : FB494_Robot_Hyundai_HMMI_v1;
    INST2 : FB494_Robot_Hyundai_HMMI_v1;
    _R102_1_1_PLT_언로딩완료 : BOOL;
END_VAR
(* ladder body could not be read *)
END_PROGRAM

PROGRAM S102_이상 (* task: 스캔 프로그램 *)
VAR
    INST10 : TON;
    INST11 : TON;
    INST12 : TON;
    INST13 : TON;
    INST14 : TON;
    INST15 : TON;
    INST16 : TON;
    INST17 : TON;
    INST18 : TON;
    INST19 : TON;
    INST20 : TON;
    INST21 : TON;
    INST22 : TON;
    INST23 : TON;
    INST24 : TON;
    INST25 : TON;
    INST26 : TON;
    INST27 : TON;
    INST28 : TON;
    INST8 : TON;
    INST9 : TON;
END_VAR
VAR_EXTERNAL
    R102_1_1_M_RB_통신이상 : BOOL; (* AT %MW1524.3 *)
    R102_1_1_M_차종3_LHD : BOOL; (* AT %MW10041.14 *) (* R102_1_1_M_차종3_LHD *)
    R102_1_1_M_차종3_RHD : BOOL; (* AT %MW10041.15 *) (* R102_1_1_M_차종3_RHD *)
    R102_1_1_M_차종5_AT : BOOL; (* AT %MW10043.1 *) (* R102_1_1_M_차종5_AT *)
    R102_1_1_M_차종5_MT : BOOL; (* AT %MW10043.0 *) (* R102_1_1_M_차종5_MT *)
    R102_1_M_RB_통신이상 : BOOL; (* AT %MW1524.4 *)
    S101_M_총괄_비상정지_이상 : BOOL; (* AT %MW1009.1 *)
    S102_6_20_PLC_BOX_CP_TRIP : BOOL; (* AT %MW86202.15 *) (* 입력 접점 15 *)
    S102_M_DASH_랙방1_2_통신이상 : BOOL; (* AT %MW1524.1 *)
    S102_M_DASH_랙방3_4_통신이상 : BOOL; (* AT %MW1524.2 *)
    S102_M_STN_DASH_로딩완료 : BOOL; (* AT %MW1501.8 *)
    S102_M_공정_간섭무 : BOOL; (* AT %MW1504.1 *)
    S102_M_공정_제품감지_ON : BOOL; (* AT %MW1501.3 *)
    S102_M_공정_통신이상 : BOOL; (* AT %MW1524.0 *)
    S102_M_사양_이상 : BOOL; (* AT %MW1516.0 *)
    S102_M_제품감지_이상 : BOOL; (* AT %MW1514.0 *)
    S102_M_차종1_AX : BOOL; (* AT %MW10061.0 *) (* S102_M_차종1_AX *)
    S102_M_총괄_CP_이상 : BOOL; (* AT %MW1509.7 *)
    S102_M_총괄_CT_이상 : BOOL; (* AT %MW1510.4 *)
    S102_M_총괄_EOCR_이상 : BOOL; (* AT %MW1509.8 *)
    S102_M_총괄_INV_이상 : BOOL; (* AT %MW1509.9 *)
    S102_M_총괄_LS_이상 : BOOL; (* AT %MW1509.15 *)
    S102_M_총괄_MATCH_이상 : BOOL; (* AT %MW1510.0 *)
    S102_M_총괄_MC_이상 : BOOL; (* AT %MW1509.13 *)
    S102_M_총괄_NFB_이상 : BOOL; (* AT %MW1509.11 *)
    S102_M_총괄_ROBOT_이상 : BOOL; (* AT %MW1510.1 *)
    S102_M_총괄_SAFETY_이상 : BOOL; (* AT %MW1509.2 *)
    S102_M_총괄_공기압_이상 : BOOL; (* AT %MW1509.3 *)
    S102_M_총괄_비상정지_이상 : BOOL; (* AT %MW1509.1 *)
    S102_M_총괄_사양_이상 : BOOL; (* AT %MW1509.6 *)
    S102_M_총괄_오버런_이상 : BOOL; (* AT %MW1509.12 *)
    S102_M_총괄_용점타점수_이상 : BOOL; (* AT %MW1510.2 *)
    S102_M_총괄_이상 : BOOL; (* AT %MW1509.0 *)
    S102_M_총괄_제품감지_이상 : BOOL; (* AT %MW1509.4 *)
    S102_M_총괄_차종_이상 : BOOL; (* AT %MW1509.5 *)
    S102_M_총괄_통신_이상 : BOOL; (* AT %MW1509.14 *)
    S102_PRS_I_AT_감지 : BOOL; (* AT %MW86201.8 *)
    S102_PRS_I_AX_파트_ON : BOOL; (* AT %MW86200.1 *)
    S102_PRS_I_LHD_감지 : BOOL; (* AT %MW86201.0 *)
    S102_PRS_I_MT_감지 : BOOL; (* AT %MW86201.9 *)
    S102_PRS_I_RHD_감지 : BOOL; (* AT %MW86201.1 *)
    S102_PRS_I_공용_파트_ON : BOOL; (* AT %MW86200.0 *)
    _0004_EB08_CFG_ER : BOOL; (* AT %MX59560 *) (* EB 구성 에러 *)
    _0004_EB08_DEER : BOOL; (* AT %MX59561 *) (* EB 운전 중 탈락 *)
    _0004_EB09_CFG_ER : BOOL; (* AT %MX59600 *) (* EB 구성 에러 *)
    _0004_EB09_DEER : BOOL; (* AT %MX59601 *) (* EB 운전 중 탈락 *)
    _0006_EB10_CFG_ER : BOOL; (* AT %MW186022.0 *) (* EB 구성 에러 *)
    _0006_EB10_DEER : BOOL; (* AT %MW186022.1 *) (* EB 운전 중 탈락 *)
    _0006_EB10_IO_DEER : BOOL; (* AT %MW186023.2 *) (* EB IO 탈락 에러 *)
    _0006_EB10_IO_TYER : BOOL; (* AT %MW186023.1 *) (* EB IO 타입 에러 *)
    _0006_EB20_CFG_ER : BOOL; (* AT %MW186028.0 *) (* EB 구성 에러 *)
    _0006_EB20_DEER : BOOL; (* AT %MW186028.1 *) (* EB 운전 중 탈락 *)
    _0006_EB20_IO_DEER : BOOL; (* AT %MW186029.2 *) (* EB IO 탈락 에러 *)
    _0006_EB20_IO_TYER : BOOL; (* AT %MW186029.1 *) (* EB IO 타입 에러 *)
    _0007_EB30_CFG_ER : BOOL; (* AT %MW187034.0 *) (* EB 구성 에러 *)
    _0007_EB30_DEER : BOOL; (* AT %MW187034.1 *) (* EB 운전 중 탈락 *)
    _0007_EB30_IO_DEER : BOOL; (* AT %MW187035.2 *) (* EB IO 탈락 에러 *)
    _0007_EB30_IO_TYER : BOOL; (* AT %MW187035.1 *) (* EB IO 타입 에러 *)
    전체_M_이상_리셋 : BOOL; (* AT %MW308.2 *) (* 전체 M 이상 리셋 *)
END_VAR

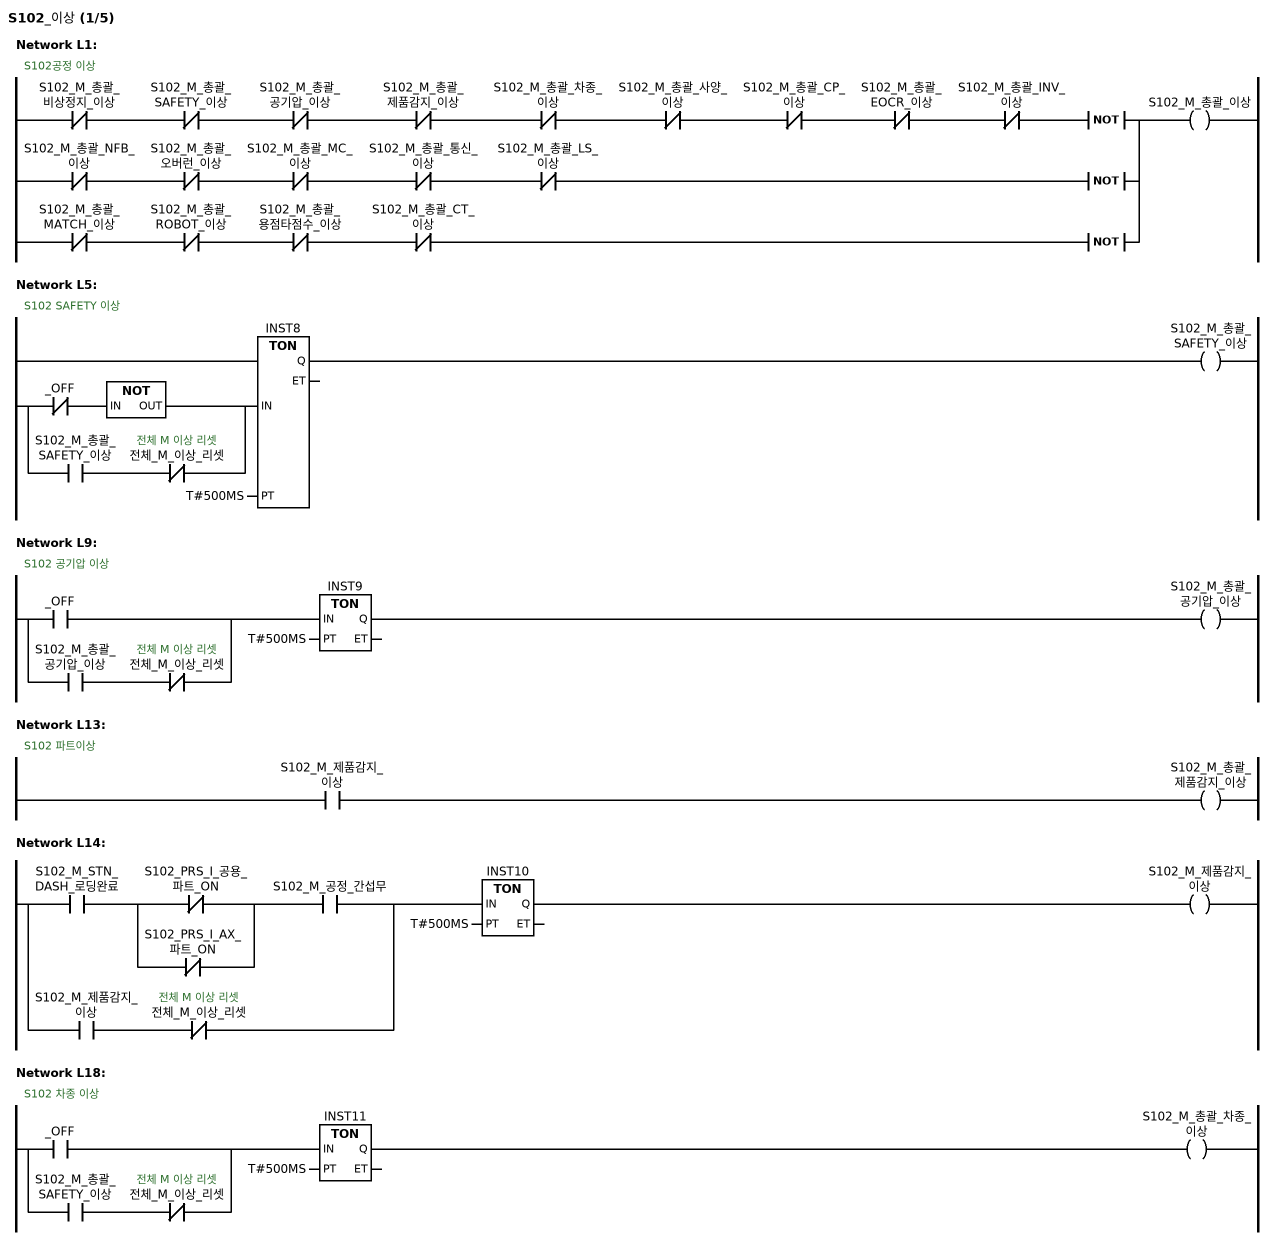
(* S102공정 이상 *)
(* Rung L1 *)
S102_M_총괄_이상 := NOT (NOT S102_M_총괄_비상정지_이상 AND NOT S102_M_총괄_SAFETY_이상 AND NOT S102_M_총괄_공기압_이상 AND NOT S102_M_총괄_제품감지_이상 AND NOT S102_M_총괄_차종_이상 AND NOT S102_M_총괄_사양_이상 AND NOT S102_M_총괄_CP_이상 AND NOT S102_M_총괄_EOCR_이상 AND NOT S102_M_총괄_INV_이상) OR NOT (NOT S102_M_총괄_NFB_이상 AND NOT S102_M_총괄_오버런_이상 AND NOT S102_M_총괄_MC_이상 AND NOT S102_M_총괄_통신_이상 AND NOT S102_M_총괄_LS_이상) OR NOT (NOT S102_M_총괄_MATCH_이상 AND NOT S102_M_총괄_ROBOT_이상 AND NOT S102_M_총괄_용점타점수_이상 AND NOT S102_M_총괄_CT_이상);
(* S102 SAFETY 이상 *)
(* Rung L5 *)
INST8(IN := (NOT (NOT _OFF)) OR (S102_M_총괄_SAFETY_이상 AND NOT 전체_M_이상_리셋), PT := T#500MS);
S102_M_총괄_SAFETY_이상 := INST8.Q;
(* S102 공기압 이상 *)
(* Rung L9 *)
INST9(IN := _OFF OR (S102_M_총괄_공기압_이상 AND NOT 전체_M_이상_리셋), PT := T#500MS);
S102_M_총괄_공기압_이상 := INST9.Q;
(* S102 파트이상 *)
(* Rung L13 *)
S102_M_총괄_제품감지_이상 := S102_M_제품감지_이상;
(* Rung L14 *)
INST10(IN := (S102_M_STN_DASH_로딩완료 AND (NOT S102_PRS_I_공용_파트_ON OR NOT S102_PRS_I_AX_파트_ON) AND S102_M_공정_간섭무) OR (S102_M_제품감지_이상 AND NOT 전체_M_이상_리셋), PT := T#500MS);
S102_M_제품감지_이상 := INST10.Q;
(* S102 차종 이상 *)
(* Rung L18 *)
INST11(IN := _OFF OR (S102_M_총괄_SAFETY_이상 AND NOT 전체_M_이상_리셋), PT := T#500MS);
S102_M_총괄_차종_이상 := INST11.Q;

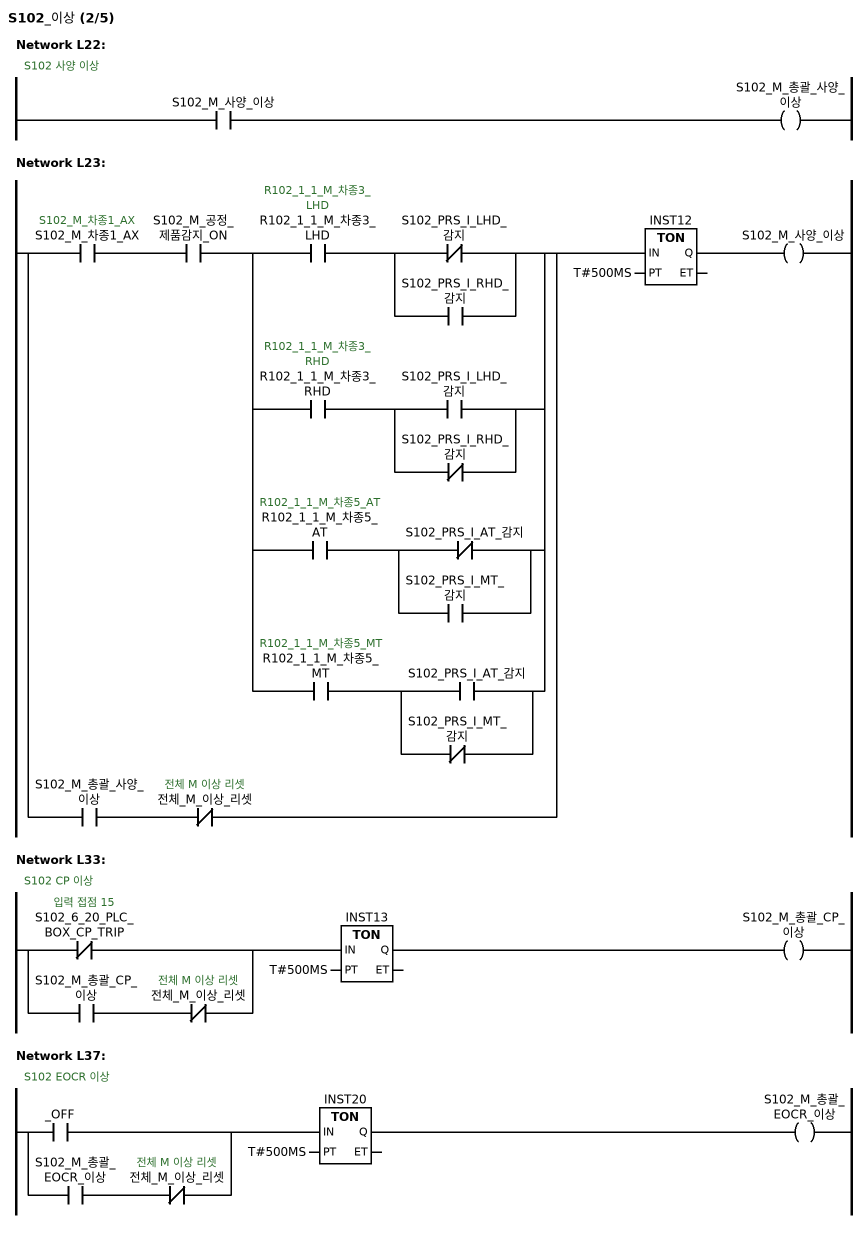
(* S102 사양 이상 *)
(* Rung L22 *)
S102_M_총괄_사양_이상 := S102_M_사양_이상;
(* Rung L23 *)
INST12(IN := (S102_M_차종1_AX AND S102_M_공정_제품감지_ON AND ((R102_1_1_M_차종3_LHD AND (NOT S102_PRS_I_LHD_감지 OR S102_PRS_I_RHD_감지)) OR (R102_1_1_M_차종3_RHD AND (S102_PRS_I_LHD_감지 OR NOT S102_PRS_I_RHD_감지)) OR (R102_1_1_M_차종5_AT AND (NOT S102_PRS_I_AT_감지 OR S102_PRS_I_MT_감지)) OR (R102_1_1_M_차종5_MT AND (S102_PRS_I_AT_감지 OR NOT S102_PRS_I_MT_감지)))) OR (S102_M_총괄_사양_이상 AND NOT 전체_M_이상_리셋), PT := T#500MS);
S102_M_사양_이상 := INST12.Q;
(* S102 CP 이상 *)
(* Rung L33 *)
INST13(IN := NOT S102_6_20_PLC_BOX_CP_TRIP OR (S102_M_총괄_CP_이상 AND NOT 전체_M_이상_리셋), PT := T#500MS);
S102_M_총괄_CP_이상 := INST13.Q;
(* S102 EOCR 이상 *)
(* Rung L37 *)
INST20(IN := _OFF OR (S102_M_총괄_EOCR_이상 AND NOT 전체_M_이상_리셋), PT := T#500MS);
S102_M_총괄_EOCR_이상 := INST20.Q;

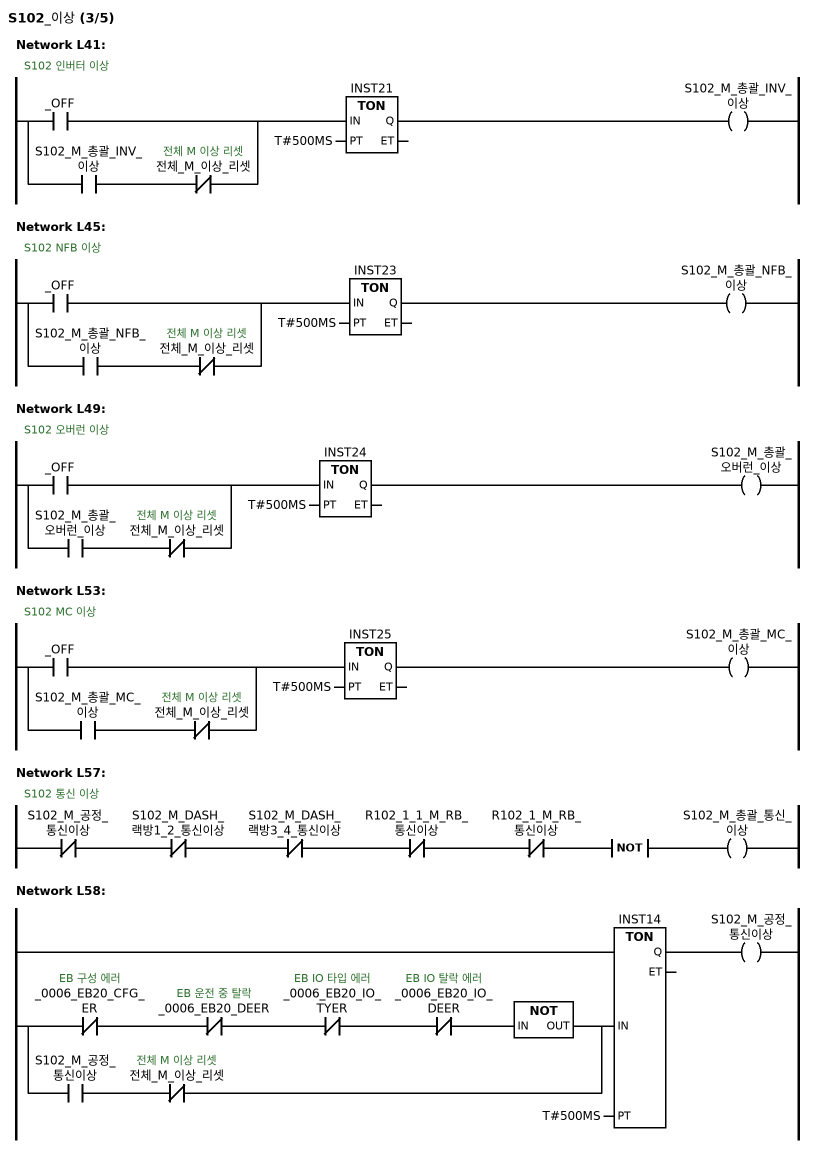
(* S102 인버터 이상 *)
(* Rung L41 *)
INST21(IN := _OFF OR (S102_M_총괄_INV_이상 AND NOT 전체_M_이상_리셋), PT := T#500MS);
S102_M_총괄_INV_이상 := INST21.Q;
(* S102 NFB 이상 *)
(* Rung L45 *)
INST23(IN := _OFF OR (S102_M_총괄_NFB_이상 AND NOT 전체_M_이상_리셋), PT := T#500MS);
S102_M_총괄_NFB_이상 := INST23.Q;
(* S102 오버런 이상 *)
(* Rung L49 *)
INST24(IN := _OFF OR (S102_M_총괄_오버런_이상 AND NOT 전체_M_이상_리셋), PT := T#500MS);
S102_M_총괄_오버런_이상 := INST24.Q;
(* S102 MC 이상 *)
(* Rung L53 *)
INST25(IN := _OFF OR (S102_M_총괄_MC_이상 AND NOT 전체_M_이상_리셋), PT := T#500MS);
S102_M_총괄_MC_이상 := INST25.Q;
(* S102 통신 이상 *)
(* Rung L57 *)
S102_M_총괄_통신_이상 := NOT (NOT S102_M_공정_통신이상 AND NOT S102_M_DASH_랙방1_2_통신이상 AND NOT S102_M_DASH_랙방3_4_통신이상 AND NOT R102_1_1_M_RB_통신이상 AND NOT R102_1_M_RB_통신이상);
(* Rung L58 *)
INST14(IN := (NOT (NOT _0006_EB20_CFG_ER AND NOT _0006_EB20_DEER AND NOT _0006_EB20_IO_TYER AND NOT _0006_EB20_IO_DEER)) OR (S102_M_공정_통신이상 AND NOT 전체_M_이상_리셋), PT := T#500MS);
S102_M_공정_통신이상 := INST14.Q;

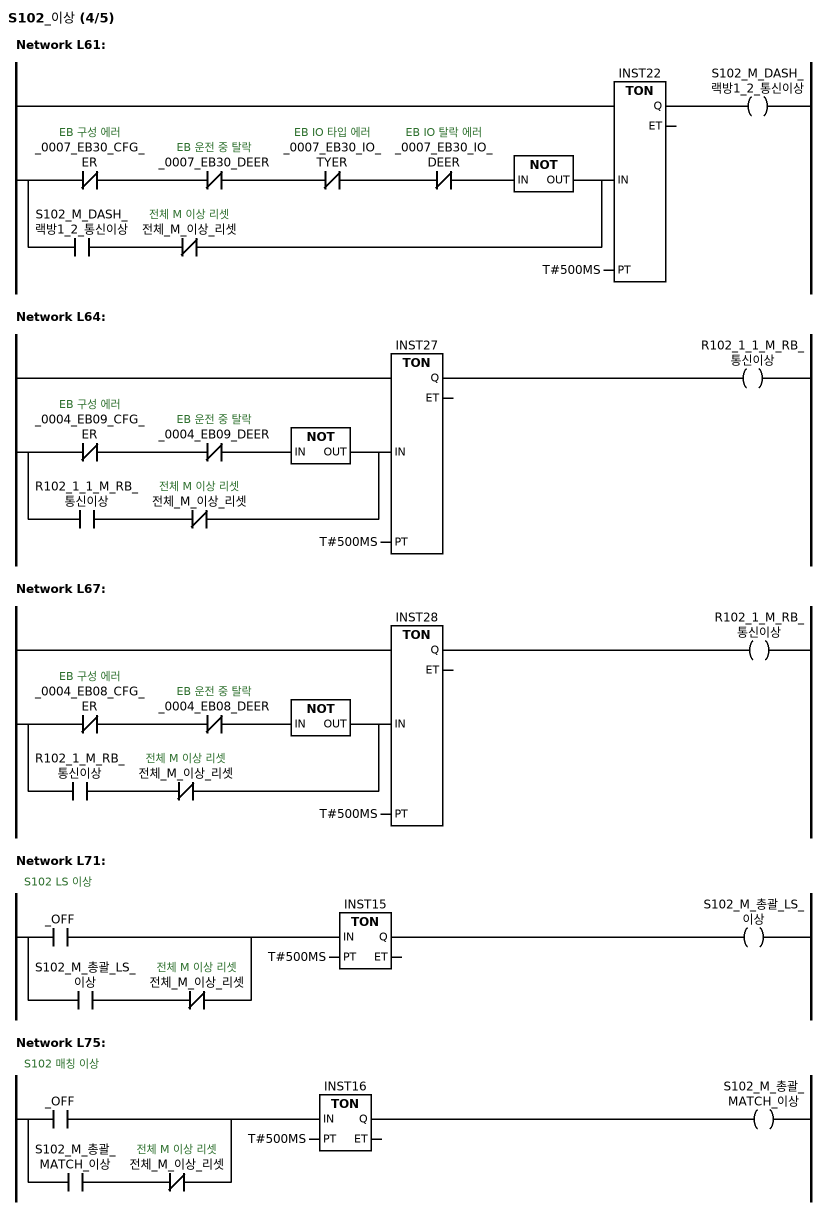
(* Rung L61 *)
INST22(IN := (NOT (NOT _0007_EB30_CFG_ER AND NOT _0007_EB30_DEER AND NOT _0007_EB30_IO_TYER AND NOT _0007_EB30_IO_DEER)) OR (S102_M_DASH_랙방1_2_통신이상 AND NOT 전체_M_이상_리셋), PT := T#500MS);
S102_M_DASH_랙방1_2_통신이상 := INST22.Q;
(* Rung L64 *)
INST27(IN := (NOT (NOT _0004_EB09_CFG_ER AND NOT _0004_EB09_DEER)) OR (R102_1_1_M_RB_통신이상 AND NOT 전체_M_이상_리셋), PT := T#500MS);
R102_1_1_M_RB_통신이상 := INST27.Q;
(* Rung L67 *)
INST28(IN := (NOT (NOT _0004_EB08_CFG_ER AND NOT _0004_EB08_DEER)) OR (R102_1_M_RB_통신이상 AND NOT 전체_M_이상_리셋), PT := T#500MS);
R102_1_M_RB_통신이상 := INST28.Q;
(* S102 LS 이상 *)
(* Rung L71 *)
INST15(IN := _OFF OR (S102_M_총괄_LS_이상 AND NOT 전체_M_이상_리셋), PT := T#500MS);
S102_M_총괄_LS_이상 := INST15.Q;
(* S102 매칭 이상 *)
(* Rung L75 *)
INST16(IN := _OFF OR (S102_M_총괄_MATCH_이상 AND NOT 전체_M_이상_리셋), PT := T#500MS);
S102_M_총괄_MATCH_이상 := INST16.Q;

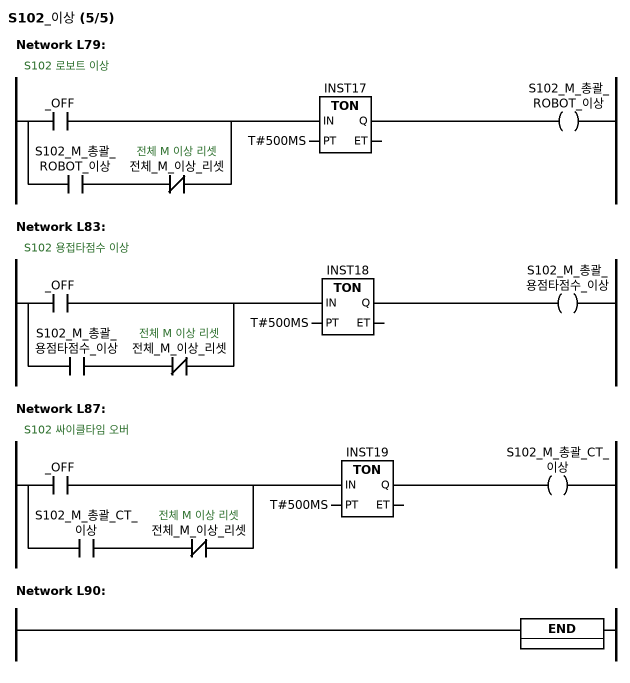
(* S102 로보트 이상 *)
(* Rung L79 *)
INST17(IN := _OFF OR (S102_M_총괄_ROBOT_이상 AND NOT 전체_M_이상_리셋), PT := T#500MS);
S102_M_총괄_ROBOT_이상 := INST17.Q;
(* S102 용접타점수 이상 *)
(* Rung L83 *)
INST18(IN := _OFF OR (S102_M_총괄_용점타점수_이상 AND NOT 전체_M_이상_리셋), PT := T#500MS);
S102_M_총괄_용점타점수_이상 := INST18.Q;
(* S102 싸이클타임 오버 *)
(* Rung L87 *)
INST19(IN := _OFF OR (S102_M_총괄_CT_이상 AND NOT 전체_M_이상_리셋), PT := T#500MS);
S102_M_총괄_CT_이상 := INST19.Q;
(* Rung L90 *)
END();
END_PROGRAM

PROGRAM S103_유틸리티 (* task: 스캔 프로그램 *)
VAR_EXTERNAL
    EGIS_EJS : BOOL;
    MCP_PBL_103_4_자동_운전 : BOOL; (* AT %MW87630.10 *) (* 입력 접점 10 *)
    MCP_PBL_운전준비_ON : BOOL; (* AT %MW87630.0 *) (* 입력 접점 00 *)
    MCP_SSP_103_4_수동_선택 : BOOL; (* AT %MW87630.8 *) (* 입력 접점 08 *)
    MCP_SSP_103_4_자동_선택 : BOOL; (* AT %MW87630.9 *) (* 입력 접점 09 *)
    R102_1_M_I_RB_간섭무_1 : BOOL; (* AT %MW20082.0 *)
    R102_1_M_I_RB_간섭무_4 : BOOL; (* AT %MW20082.3 *)
    R102_1_M_I_RB_원위치 : BOOL; (* AT %MW20080.3 *)
    R103_1_M_I_RB_간섭무_1 : BOOL; (* AT %MW20102.0 *)
    R103_1_M_I_RB_간섭무_4 : BOOL; (* AT %MW20102.3 *)
    R103_1_M_I_RB_원위치 : BOOL; (* AT %MW20100.3 *)
    R103_1_M_SEQ : WORD; (* AT %MW10120 *) (* R103_1_M_SEQ *)
    R103_1_M_STN_차종_NONE : BOOL; (* AT %MW2002.3 *)
    R103_1_M_STN_차종_ON : BOOL; (* AT %MW2002.2 *)
    R103_1_M_차종1_AX : BOOL; (* AT %MW10121.0 *) (* R103_1_M_차종1_AX *)
    R103_1_M_차종1_B : BOOL; (* AT %MW10121.1 *) (* R103_1_M_차종1_B *)
    R103_1_M_차종1_C : BOOL; (* AT %MW10121.2 *) (* R103_1_M_차종1_C *)
    R103_1_M_차종1_D : BOOL; (* AT %MW10121.3 *) (* R103_1_M_차종1_D *)
    R103_1_M_차종1_E : BOOL; (* AT %MW10121.4 *) (* R103_1_M_차종1_E *)
    R103_1_M_차종1_F : BOOL; (* AT %MW10121.5 *) (* R103_1_M_차종1_F *)
    R103_1_M_차종1_G : BOOL; (* AT %MW10121.6 *) (* R103_1_M_차종1_G *)
    R103_1_M_차종1_H : BOOL; (* AT %MW10121.7 *) (* R103_1_M_차종1_H *)
    R103_1_M_차종2_3DR : BOOL; (* AT %MW10121.8 *) (* R103_1_M_차종2_3DR *)
    R103_1_M_차종2_4DR : BOOL; (* AT %MW10121.9 *) (* R103_1_M_차종2_4DR *)
    R103_1_M_차종2_5DR : BOOL; (* AT %MW10121.10 *) (* R103_1_M_차종2_5DR *)
    R103_1_M_차종2_SP1 : BOOL; (* AT %MW10121.12 *) (* R103_1_M_차종2_SP1 *)
    R103_1_M_차종2_SP2 : BOOL; (* AT %MW10121.13 *) (* R103_1_M_차종2_SP2 *)
    R103_1_M_차종2_WGN : BOOL; (* AT %MW10121.11 *) (* R103_1_M_차종2_WGN *)
    R103_1_M_차종3_LHD : BOOL; (* AT %MW10121.14 *) (* R103_1_M_차종3_LHD *)
    R103_1_M_차종3_RHD : BOOL; (* AT %MW10121.15 *) (* R103_1_M_차종3_RHD *)
    R103_1_M_차종4_EEC : BOOL; (* AT %MW10122.3 *) (* R103_1_M_차종4_EEC *)
    R103_1_M_차종4_SP1 : BOOL; (* AT %MW10122.8 *) (* R103_1_M_차종4_SP1 *)
    R103_1_M_차종4_SP2 : BOOL; (* AT %MW10122.9 *) (* R103_1_M_차종4_SP2 *)
    R103_1_M_차종4_SP3 : BOOL; (* AT %MW10122.11 *) (* R103_1_M_차종4_SP3 *)
    R103_1_M_차종4_SP4 : BOOL; (* AT %MW10122.12 *) (* R103_1_M_차종4_SP4 *)
    R103_1_M_차종4_SP5 : BOOL; (* AT %MW10122.13 *) (* R103_1_M_차종4_SP5 *)
    R103_1_M_차종4_SP6 : BOOL; (* AT %MW10122.14 *) (* R103_1_M_차종4_SP6 *)
    R103_1_M_차종4_SP7 : BOOL; (* AT %MW10122.15 *) (* R103_1_M_차종4_SP7 *)
    R103_1_M_차종4_내수 : BOOL; (* AT %MW10122.0 *) (* R103_1_M_차종4_내수 *)
    R103_1_M_차종4_러시아 : BOOL; (* AT %MW10122.10 *) (* R103_1_M_차종4_러시아 *)
    R103_1_M_차종4_북미 : BOOL; (* AT %MW10122.2 *) (* R103_1_M_차종4_북미 *)
    R103_1_M_차종4_브라질 : BOOL; (* AT %MW10122.7 *) (* R103_1_M_차종4_브라질 *)
    R103_1_M_차종4_수출 : BOOL; (* AT %MW10122.1 *) (* R103_1_M_차종4_수출 *)
    R103_1_M_차종4_중국 : BOOL; (* AT %MW10122.6 *) (* R103_1_M_차종4_중국 *)
    R103_1_M_차종4_중동 : BOOL; (* AT %MW10122.5 *) (* R103_1_M_차종4_중동 *)
    R103_1_M_차종4_호주 : BOOL; (* AT %MW10122.4 *) (* R103_1_M_차종4_호주 *)
    R103_1_M_차종5_AT : BOOL; (* AT %MW10123.1 *) (* R103_1_M_차종5_AT *)
    R103_1_M_차종5_MT : BOOL; (* AT %MW10123.0 *) (* R103_1_M_차종5_MT *)
    R103_1_M_차종5_SP1 : BOOL; (* AT %MW10123.2 *) (* R103_1_M_차종5_SP1 *)
    R103_1_M_차종6_DSROOF : BOOL; (* AT %MW10123.6 *) (* R103_1_M_차종6_DSROOF *)
    R103_1_M_차종6_SP1 : BOOL; (* AT %MW10123.7 *) (* R103_1_M_차종6_SP1 *)
    R103_1_M_차종6_썬루프 : BOOL; (* AT %MW10123.4 *) (* R103_1_M_차종6_썬루프 *)
    R103_1_M_차종6_일반루프 : BOOL; (* AT %MW10123.3 *) (* R103_1_M_차종6_일반루프 *)
    R103_1_M_차종6_파노라마루프 : BOOL; (* AT %MW10123.5 *) (* R103_1_M_차종6_파노라마루프 *)
    R103_1_M_차종7_DSL : BOOL; (* AT %MW10123.9 *) (* R103_1_M_차종7_DSL *)
    R103_1_M_차종7_GSL : BOOL; (* AT %MW10123.8 *) (* R103_1_M_차종7_GSL *)
    R103_1_M_차종7_SP1 : BOOL; (* AT %MW10123.10 *) (* R103_1_M_차종7_SP1 *)
    R103_1_M_차종7_SP2 : BOOL; (* AT %MW10123.11 *) (* R103_1_M_차종7_SP2 *)
    R103_1_M_차종7_SP3 : BOOL; (* AT %MW10123.12 *) (* R103_1_M_차종7_SP3 *)
    R103_1_M_차종7_SP4 : BOOL; (* AT %MW10123.13 *) (* R103_1_M_차종7_SP4 *)
    R103_1_M_차종7_SP5 : BOOL; (* AT %MW10123.14 *) (* R103_1_M_차종7_SP5 *)
    R103_1_M_차종7_SP6 : BOOL; (* AT %MW10123.15 *) (* R103_1_M_차종7_SP6 *)
    R103_1_M_차종8_2WD : BOOL; (* AT %MW10124.0 *) (* R103_1_M_차종8_2WD *)
    R103_1_M_차종8_4WD : BOOL; (* AT %MW10124.1 *) (* R103_1_M_차종8_4WD *)
    R103_1_M_차종8_SP1 : BOOL; (* AT %MW10124.2 *) (* R103_1_M_차종8_SP1 *)
    R103_1_M_차종9_MPI : BOOL; (* AT %MW10124.3 *) (* R103_1_M_차종9_MPI *)
    R103_1_M_차종9_SP1 : BOOL; (* AT %MW10124.5 *) (* R103_1_M_차종9_SP1 *)
    R103_1_M_차종9_SP10 : BOOL; (* AT %MW10124.14 *) (* R103_1_M_차종9_SP10 *)
    R103_1_M_차종9_SP11 : BOOL; (* AT %MW10124.15 *) (* R103_1_M_차종9_SP11 *)
    R103_1_M_차종9_SP2 : BOOL; (* AT %MW10124.6 *) (* R103_1_M_차종9_SP2 *)
    R103_1_M_차종9_SP3 : BOOL; (* AT %MW10124.7 *) (* R103_1_M_차종9_SP3 *)
    R103_1_M_차종9_SP4 : BOOL; (* AT %MW10124.8 *) (* R103_1_M_차종9_SP4 *)
    R103_1_M_차종9_SP5 : BOOL; (* AT %MW10124.9 *) (* R103_1_M_차종9_SP5 *)
    R103_1_M_차종9_SP6 : BOOL; (* AT %MW10124.10 *) (* R103_1_M_차종9_SP6 *)
    R103_1_M_차종9_SP7 : BOOL; (* AT %MW10124.11 *) (* R103_1_M_차종9_SP7 *)
    R103_1_M_차종9_SP8 : BOOL; (* AT %MW10124.12 *) (* R103_1_M_차종9_SP8 *)
    R103_1_M_차종9_SP9 : BOOL; (* AT %MW10124.13 *) (* R103_1_M_차종9_SP9 *)
    R103_1_M_차종9_T_GDI : BOOL; (* AT %MW10124.4 *) (* R103_1_M_차종9_T_GDI *)
    R103_1_M_차종_OPT1_R_RACK_무 : BOOL; (* AT %MW10125.3 *) (* R103_1_M_차종_OPT1_R_RACK_무 *)
    R103_1_M_차종_OPT1_R_RACK_유 : BOOL; (* AT %MW10125.2 *) (* R103_1_M_차종_OPT1_R_RACK_유 *)
    R103_1_M_차종_OPT1_SP1 : BOOL; (* AT %MW10125.10 *) (* R103_1_M_차종_OPT1_SP1 *)
    R103_1_M_차종_OPT1_SP2 : BOOL; (* AT %MW10125.11 *) (* R103_1_M_차종_OPT1_SP2 *)
    R103_1_M_차종_OPT1_SP3 : BOOL; (* AT %MW10125.12 *) (* R103_1_M_차종_OPT1_SP3 *)
    R103_1_M_차종_OPT1_SP4 : BOOL; (* AT %MW10125.13 *) (* R103_1_M_차종_OPT1_SP4 *)
    R103_1_M_차종_OPT1_SP5 : BOOL; (* AT %MW10125.14 *) (* R103_1_M_차종_OPT1_SP5 *)
    R103_1_M_차종_OPT1_SP6 : BOOL; (* AT %MW10125.15 *) (* R103_1_M_차종_OPT1_SP6 *)
    R103_1_M_차종_OPT1_S_REP_EATER_무 : BOOL; (* AT %MW10125.7 *) (* R103_1_M_차종_OPT1_S_REP_EATER_무 *)
    R103_1_M_차종_OPT1_S_REP_EATER_유 : BOOL; (* AT %MW10125.6 *) (* R103_1_M_차종_OPT1_S_REP_EATER_유 *)
    R103_1_M_차종_OPT1_VAN_무 : BOOL; (* AT %MW10125.9 *) (* R103_1_M_차종_OPT1_VAN_무 *)
    R103_1_M_차종_OPT1_VAN_유 : BOOL; (* AT %MW10125.8 *) (* R103_1_M_차종_OPT1_VAN_유 *)
    R103_1_M_차종_OPT1_슬라이딩_무 : BOOL; (* AT %MW10125.1 *) (* R103_1_M_차종_OPT1_슬라이딩_무 *)
    R103_1_M_차종_OPT1_슬라이딩_유 : BOOL; (* AT %MW10125.0 *) (* R103_1_M_차종_OPT1_슬라이딩_유 *)
    R103_1_M_차종_OPT1_폴딩_무 : BOOL; (* AT %MW10125.5 *) (* R103_1_M_차종_OPT1_폴딩_무 *)
    R103_1_M_차종_OPT1_폴딩_유 : BOOL; (* AT %MW10125.4 *) (* R103_1_M_차종_OPT1_폴딩_유 *)
    S102_M_작업_완료 : BOOL; (* AT %MW1501.0 *)
    S103_M_AX_래치_전진단 : BOOL; (* AT %MW2100.3 *)
    S103_M_AX_래치_후진단 : BOOL; (* AT %MW2100.4 *)
    S103_M_SEQ : WORD; (* AT %MW10100 *) (* S103_M_SEQ *)
    S103_M_STN_차종_NONE : BOOL; (* AT %MW2002.1 *)
    S103_M_STN_차종_ON : BOOL; (* AT %MW2002.0 *)
    S103_M_공정_HOME_POSI : BOOL; (* AT %MW2004.0 *)
    S103_M_공정_간섭무 : BOOL; (* AT %MW2004.1 *)
    S103_M_공정_제품감지_OFF : BOOL; (* AT %MW2001.4 *)
    S103_M_공정_제품감지_ON : BOOL; (* AT %MW2001.3 *)
    S103_M_수동_모드 : BOOL; (* AT %MW2000.3 *)
    S103_M_운전준비_ON : BOOL; (* AT %MW2000.0 *)
    S103_M_자동_START : BOOL; (* AT %MW2000.5 *)
    S103_M_자동_모드 : BOOL; (* AT %MW2000.1 *)
    S103_M_자동_운전중 : BOOL; (* AT %MW2000.4 *)
    S103_M_작업_완료 : BOOL; (* AT %MW2001.0 *)
    S103_M_작업_완료_보조 : BOOL; (* AT %MW2000.9 *)
    S103_M_차종1_AX : BOOL; (* AT %MW10101.0 *) (* S103_M_차종1_AX *)
    S103_M_차종1_B : BOOL; (* AT %MW10101.1 *) (* S103_M_차종1_B *)
    S103_M_차종1_C : BOOL; (* AT %MW10101.2 *) (* S103_M_차종1_C *)
    S103_M_차종1_D : BOOL; (* AT %MW10101.3 *) (* S103_M_차종1_D *)
    S103_M_차종1_E : BOOL; (* AT %MW10101.4 *) (* S103_M_차종1_E *)
    S103_M_차종1_F : BOOL; (* AT %MW10101.5 *) (* S103_M_차종1_F *)
    S103_M_차종1_G : BOOL; (* AT %MW10101.6 *) (* S103_M_차종1_G *)
    S103_M_차종1_H : BOOL; (* AT %MW10101.7 *) (* S103_M_차종1_H *)
    S103_M_차종2_3DR : BOOL; (* AT %MW10101.8 *) (* S103_M_차종2_3DR *)
    S103_M_차종2_4DR : BOOL; (* AT %MW10101.9 *) (* S103_M_차종2_4DR *)
    S103_M_차종2_5DR : BOOL; (* AT %MW10101.10 *) (* S103_M_차종2_5DR *)
    S103_M_차종2_SP1 : BOOL; (* AT %MW10101.12 *) (* S103_M_차종2_SP1 *)
    S103_M_차종2_SP2 : BOOL; (* AT %MW10101.13 *) (* S103_M_차종2_SP2 *)
    S103_M_차종2_WGN : BOOL; (* AT %MW10101.11 *) (* S103_M_차종2_WGN *)
    S103_M_차종3_LHD : BOOL; (* AT %MW10101.14 *) (* S103_M_차종3_LHD *)
    S103_M_차종3_RHD : BOOL; (* AT %MW10101.15 *) (* S103_M_차종3_RHD *)
    S103_M_차종4_EEC : BOOL; (* AT %MW10102.3 *) (* S103_M_차종4_EEC *)
    S103_M_차종4_SP1 : BOOL; (* AT %MW10102.8 *) (* S103_M_차종4_SP1 *)
    S103_M_차종4_SP2 : BOOL; (* AT %MW10102.9 *) (* S103_M_차종4_SP2 *)
    S103_M_차종4_SP3 : BOOL; (* AT %MW10102.11 *) (* S103_M_차종4_SP3 *)
    S103_M_차종4_SP4 : BOOL; (* AT %MW10102.12 *) (* S103_M_차종4_SP4 *)
    S103_M_차종4_SP5 : BOOL; (* AT %MW10102.13 *) (* S103_M_차종4_SP5 *)
    S103_M_차종4_SP6 : BOOL; (* AT %MW10102.14 *) (* S103_M_차종4_SP6 *)
    S103_M_차종4_SP7 : BOOL; (* AT %MW10102.15 *) (* S103_M_차종4_SP7 *)
    S103_M_차종4_내수 : BOOL; (* AT %MW10102.0 *) (* S103_M_차종4_내수 *)
    S103_M_차종4_러시아 : BOOL; (* AT %MW10102.10 *) (* S103_M_차종4_러시아 *)
    S103_M_차종4_북미 : BOOL; (* AT %MW10102.2 *) (* S103_M_차종4_북미 *)
    S103_M_차종4_브라질 : BOOL; (* AT %MW10102.7 *) (* S103_M_차종4_브라질 *)
    S103_M_차종4_수출 : BOOL; (* AT %MW10102.1 *) (* S103_M_차종4_수출 *)
    S103_M_차종4_중국 : BOOL; (* AT %MW10102.6 *) (* S103_M_차종4_중국 *)
    S103_M_차종4_중동 : BOOL; (* AT %MW10102.5 *) (* S103_M_차종4_중동 *)
    S103_M_차종4_호주 : BOOL; (* AT %MW10102.4 *) (* S103_M_차종4_호주 *)
    S103_M_차종5_AT : BOOL; (* AT %MW10103.1 *) (* S103_M_차종5_AT *)
    S103_M_차종5_MT : BOOL; (* AT %MW10103.0 *) (* S103_M_차종5_MT *)
    S103_M_차종5_SP1 : BOOL; (* AT %MW10103.2 *) (* S103_M_차종5_SP1 *)
    S103_M_차종6_DSROOF : BOOL; (* AT %MW10103.6 *) (* S103_M_차종6_DSROOF *)
    S103_M_차종6_SP1 : BOOL; (* AT %MW10103.7 *) (* S103_M_차종6_SP1 *)
    S103_M_차종6_썬루프 : BOOL; (* AT %MW10103.4 *) (* S103_M_차종6_썬루프 *)
    S103_M_차종6_일반루프 : BOOL; (* AT %MW10103.3 *) (* S103_M_차종6_일반루프 *)
    S103_M_차종6_파노라마루프 : BOOL; (* AT %MW10103.5 *) (* S103_M_차종6_파노라마루프 *)
    S103_M_차종7_DSL : BOOL; (* AT %MW10103.9 *) (* S103_M_차종7_DSL *)
    S103_M_차종7_GSL : BOOL; (* AT %MW10103.8 *) (* S103_M_차종7_GSL *)
    S103_M_차종7_SP1 : BOOL; (* AT %MW10103.10 *) (* S103_M_차종7_SP1 *)
    S103_M_차종7_SP2 : BOOL; (* AT %MW10103.11 *) (* S103_M_차종7_SP2 *)
    S103_M_차종7_SP3 : BOOL; (* AT %MW10103.12 *) (* S103_M_차종7_SP3 *)
    S103_M_차종7_SP4 : BOOL; (* AT %MW10103.13 *) (* S103_M_차종7_SP4 *)
    S103_M_차종7_SP5 : BOOL; (* AT %MW10103.14 *) (* S103_M_차종7_SP5 *)
    S103_M_차종7_SP6 : BOOL; (* AT %MW10103.15 *) (* S103_M_차종7_SP6 *)
    S103_M_차종8_2WD : BOOL; (* AT %MW10104.0 *) (* S103_M_차종8_2WD *)
    S103_M_차종8_4WD : BOOL; (* AT %MW10104.1 *) (* S103_M_차종8_4WD *)
    S103_M_차종8_SP1 : BOOL; (* AT %MW10104.2 *) (* S103_M_차종8_SP1 *)
    S103_M_차종9_MPI : BOOL; (* AT %MW10104.3 *) (* S103_M_차종9_MPI *)
    S103_M_차종9_SP1 : BOOL; (* AT %MW10104.5 *) (* S103_M_차종9_SP1 *)
    S103_M_차종9_SP10 : BOOL; (* AT %MW10104.14 *) (* S103_M_차종9_SP10 *)
    S103_M_차종9_SP11 : BOOL; (* AT %MW10104.15 *) (* S103_M_차종9_SP11 *)
    S103_M_차종9_SP2 : BOOL; (* AT %MW10104.6 *) (* S103_M_차종9_SP2 *)
    S103_M_차종9_SP3 : BOOL; (* AT %MW10104.7 *) (* S103_M_차종9_SP3 *)
    S103_M_차종9_SP4 : BOOL; (* AT %MW10104.8 *) (* S103_M_차종9_SP4 *)
    S103_M_차종9_SP5 : BOOL; (* AT %MW10104.9 *) (* S103_M_차종9_SP5 *)
    S103_M_차종9_SP6 : BOOL; (* AT %MW10104.10 *) (* S103_M_차종9_SP6 *)
    S103_M_차종9_SP7 : BOOL; (* AT %MW10104.11 *) (* S103_M_차종9_SP7 *)
    S103_M_차종9_SP8 : BOOL; (* AT %MW10104.12 *) (* S103_M_차종9_SP8 *)
    S103_M_차종9_SP9 : BOOL; (* AT %MW10104.13 *) (* S103_M_차종9_SP9 *)
    S103_M_차종9_T_GDI : BOOL; (* AT %MW10104.4 *) (* S103_M_차종9_T_GDI *)
    S103_M_차종_OPT1_R_RACK_무 : BOOL; (* AT %MW10105.3 *) (* S103_M_차종_OPT1_R_RACK_무 *)
    S103_M_차종_OPT1_R_RACK_유 : BOOL; (* AT %MW10105.2 *) (* S103_M_차종_OPT1_R_RACK_유 *)
    S103_M_차종_OPT1_SP1 : BOOL; (* AT %MW10105.10 *) (* S103_M_차종_OPT1_SP1 *)
    S103_M_차종_OPT1_SP2 : BOOL; (* AT %MW10105.11 *) (* S103_M_차종_OPT1_SP2 *)
    S103_M_차종_OPT1_SP3 : BOOL; (* AT %MW10105.12 *) (* S103_M_차종_OPT1_SP3 *)
    S103_M_차종_OPT1_SP4 : BOOL; (* AT %MW10105.13 *) (* S103_M_차종_OPT1_SP4 *)
    S103_M_차종_OPT1_SP5 : BOOL; (* AT %MW10105.14 *) (* S103_M_차종_OPT1_SP5 *)
    S103_M_차종_OPT1_SP6 : BOOL; (* AT %MW10105.15 *) (* S103_M_차종_OPT1_SP6 *)
    S103_M_차종_OPT1_S_REP_EATER_무 : BOOL; (* AT %MW10105.7 *) (* S103_M_차종_OPT1_S_REP_EATER_무 *)
    S103_M_차종_OPT1_S_REP_EATER_유 : BOOL; (* AT %MW10105.6 *) (* S103_M_차종_OPT1_S_REP_EATER_유 *)
    S103_M_차종_OPT1_VAN_무 : BOOL; (* AT %MW10105.9 *) (* S103_M_차종_OPT1_VAN_무 *)
    S103_M_차종_OPT1_VAN_유 : BOOL; (* AT %MW10105.8 *) (* S103_M_차종_OPT1_VAN_유 *)
    S103_M_차종_OPT1_슬라이딩_무 : BOOL; (* AT %MW10105.1 *) (* S103_M_차종_OPT1_슬라이딩_무 *)
    S103_M_차종_OPT1_슬라이딩_유 : BOOL; (* AT %MW10105.0 *) (* S103_M_차종_OPT1_슬라이딩_유 *)
    S103_M_차종_OPT1_폴딩_무 : BOOL; (* AT %MW10105.5 *) (* S103_M_차종_OPT1_폴딩_무 *)
    S103_M_차종_OPT1_폴딩_유 : BOOL; (* AT %MW10105.4 *) (* S103_M_차종_OPT1_폴딩_유 *)
    S103_PRS_AX_제품감지_CHECK1 : BOOL; (* AT %MW86301.0 *) (* 입력 접점 00 *)
    S103_PRS_AX_제품감지_CHECK2 : BOOL; (* AT %MW86301.1 *) (* 입력 접점 01 *)
    S103_운전준비 : TON;
    T103_자동 : TON;
    전체_M_GATE_자동기동 : BOOL; (* AT %MW308.1 *) (* 전체 M GATE 자동기동 *)
    전체_라인_M_총괄_SAFETY_이상 : BOOL; (* AT %MW300.2 *)
    전체_라인_M_총괄_공기압_이상 : BOOL; (* AT %MW300.3 *)
    전체_라인_M_총괄_비상정지_이상 : BOOL; (* AT %MW300.1 *)
    전체_라인_M_총괄_이상 : BOOL; (* AT %MW300.0 *)
END_VAR
VAR
    _t1 : BOOL;
    _t2 : BOOL;
END_VAR

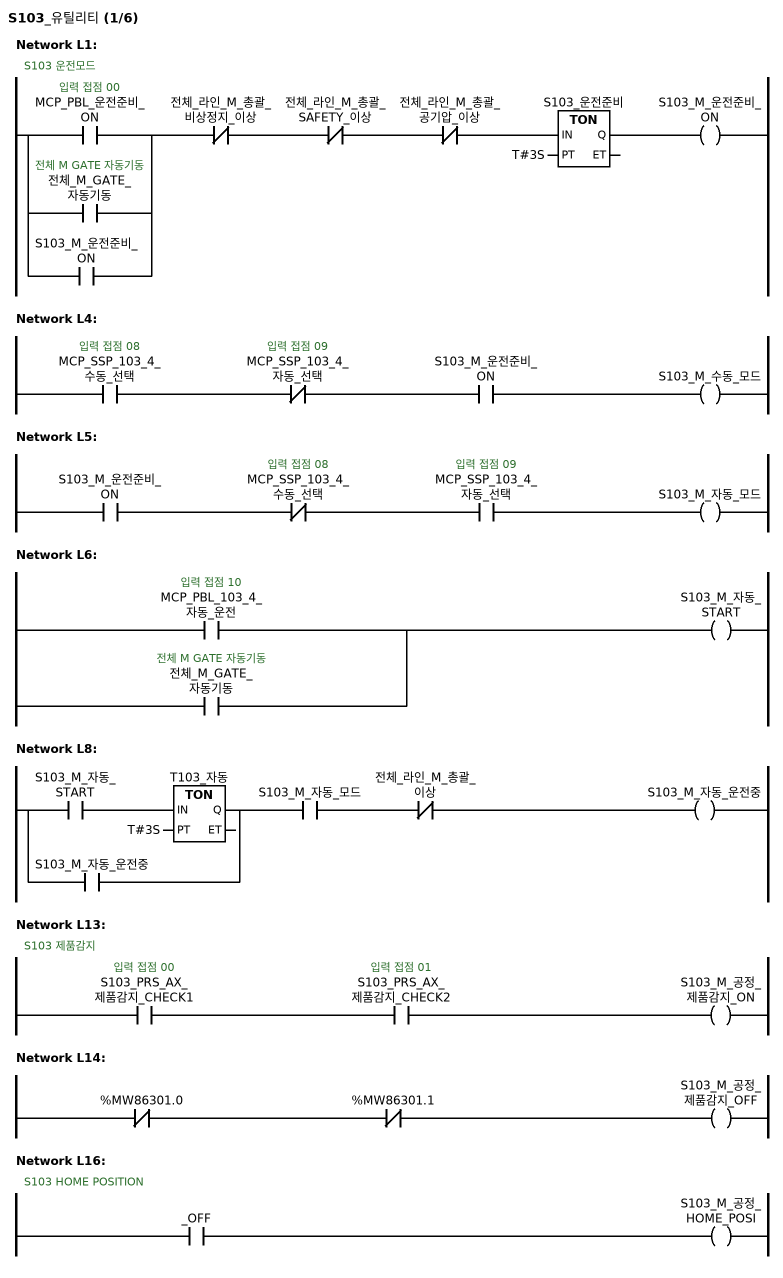
(* S103 운전모드 *)
(* Rung L1 *)
S103_운전준비(IN := (MCP_PBL_운전준비_ON OR 전체_M_GATE_자동기동 OR S103_M_운전준비_ON) AND NOT 전체_라인_M_총괄_비상정지_이상 AND NOT 전체_라인_M_총괄_SAFETY_이상 AND NOT 전체_라인_M_총괄_공기압_이상, PT := T#3S);
S103_M_운전준비_ON := S103_운전준비.Q;
(* Rung L4 *)
S103_M_수동_모드 := MCP_SSP_103_4_수동_선택 AND NOT MCP_SSP_103_4_자동_선택 AND S103_M_운전준비_ON;
(* Rung L5 *)
S103_M_자동_모드 := S103_M_운전준비_ON AND NOT MCP_SSP_103_4_수동_선택 AND MCP_SSP_103_4_자동_선택;
(* Rung L6 *)
S103_M_자동_START := MCP_PBL_103_4_자동_운전 OR 전체_M_GATE_자동기동;
(* Rung L8 *)
T103_자동(IN := S103_M_자동_START, PT := T#3S);
S103_M_자동_운전중 := (T103_자동.Q OR S103_M_자동_운전중) AND S103_M_자동_모드 AND NOT 전체_라인_M_총괄_이상;
(* S103 제품감지 *)
(* Rung L13 *)
S103_M_공정_제품감지_ON := S103_PRS_AX_제품감지_CHECK1 AND S103_PRS_AX_제품감지_CHECK2;
(* Rung L14 *)
S103_M_공정_제품감지_OFF := NOT %MW86301.0 AND NOT %MW86301.1;
(* S103 HOME POSITION *)
(* Rung L16 *)
S103_M_공정_HOME_POSI := _OFF;

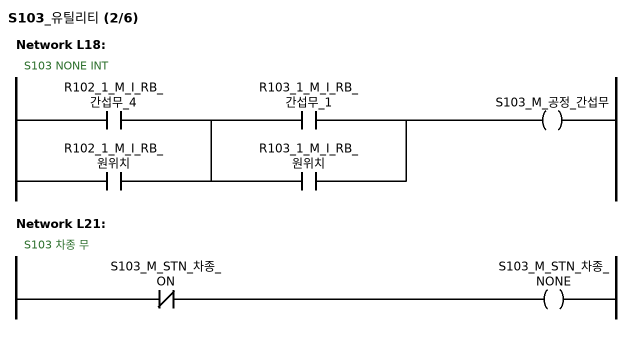
(* S103 NONE INT *)
(* Rung L18 *)
S103_M_공정_간섭무 := (R102_1_M_I_RB_간섭무_4 OR R102_1_M_I_RB_원위치) AND (R103_1_M_I_RB_간섭무_1 OR R103_1_M_I_RB_원위치);
(* S103 차종 무 *)
(* Rung L21 *)
S103_M_STN_차종_NONE := NOT S103_M_STN_차종_ON;

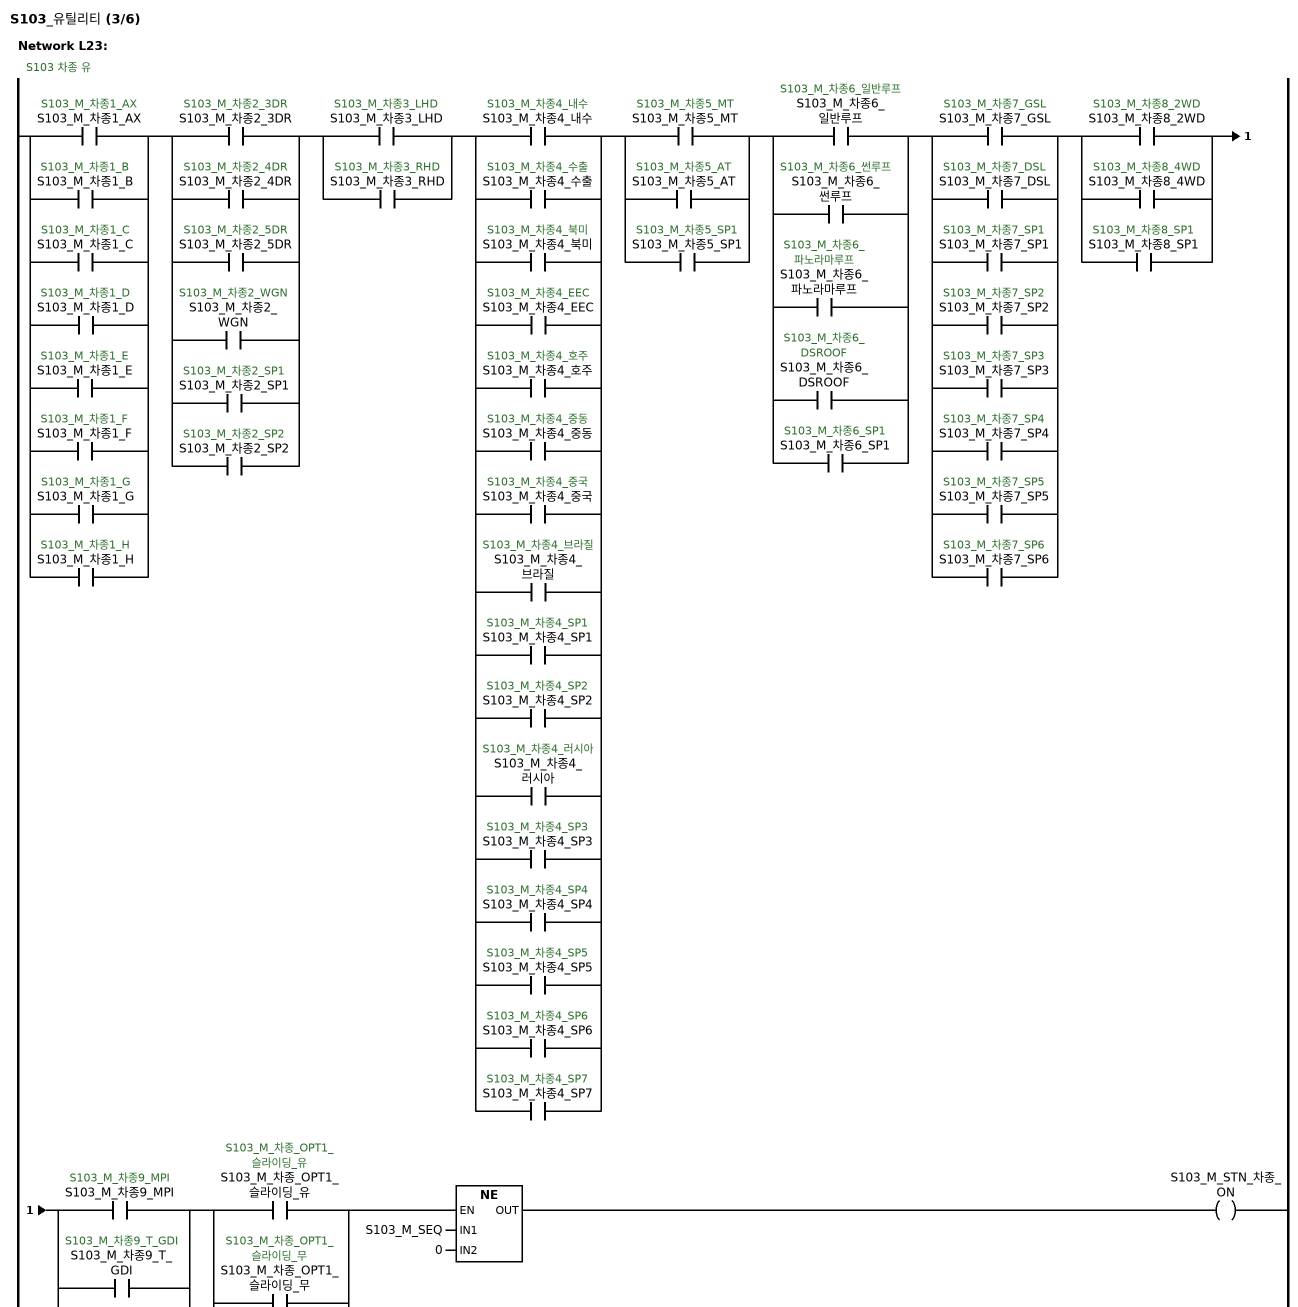

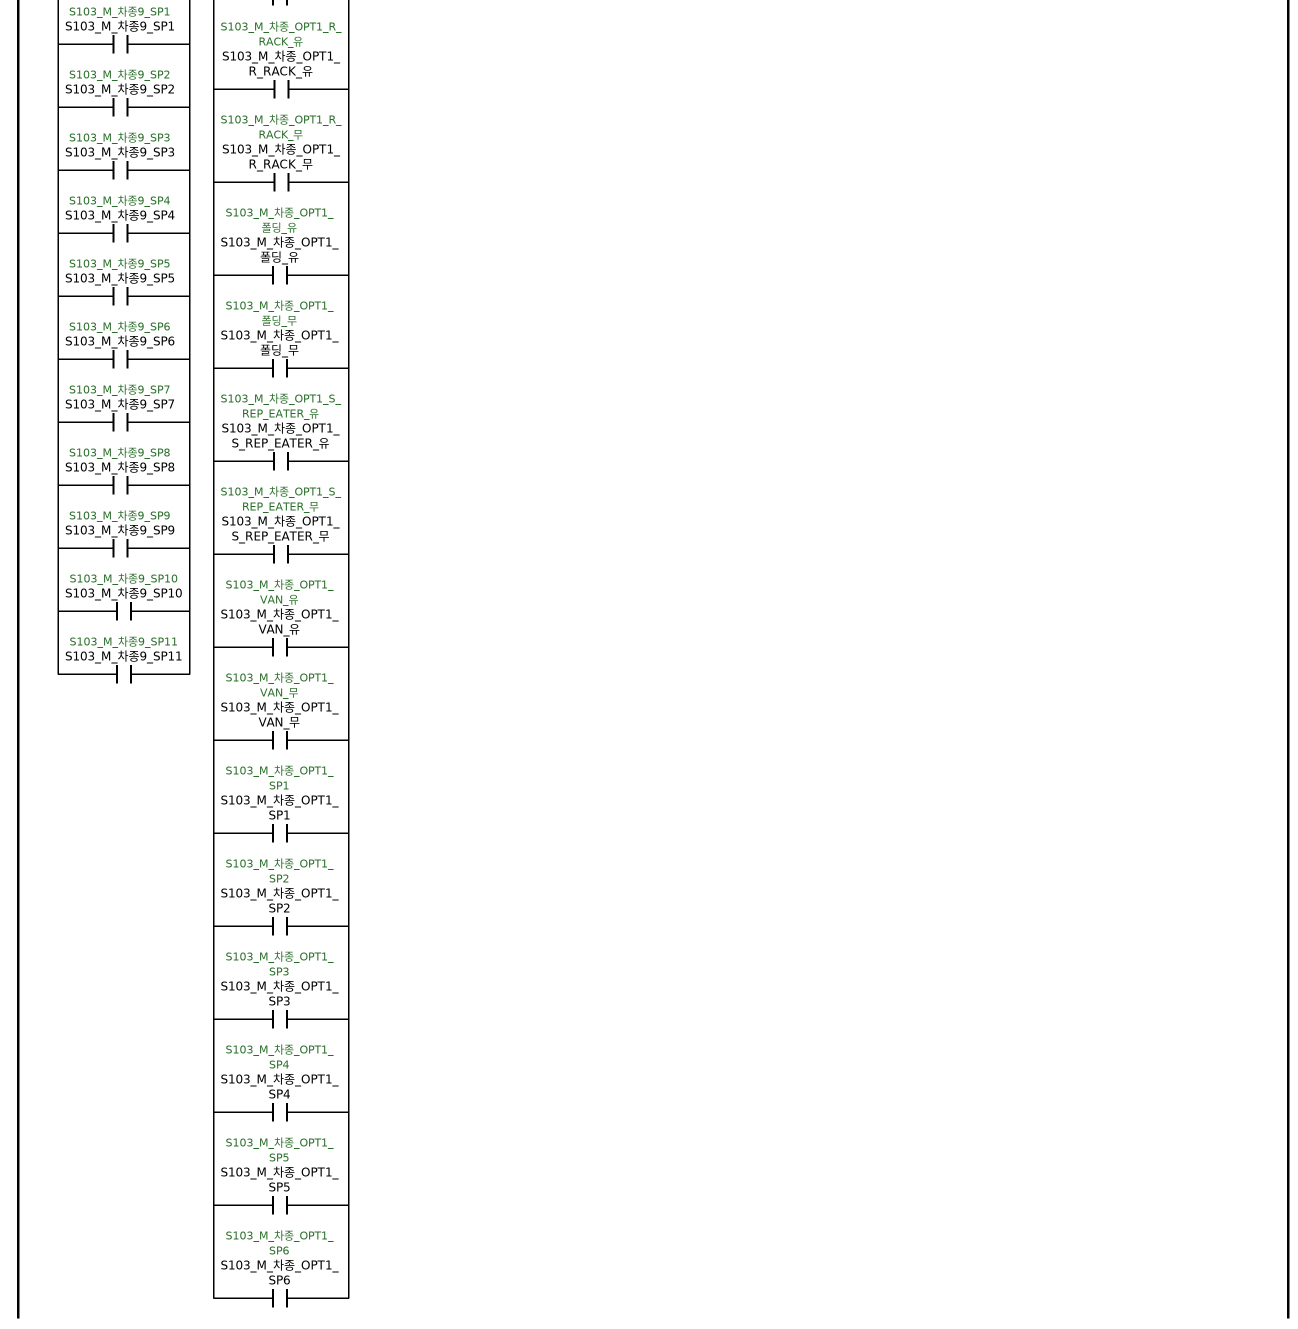
(* S103 차종 유 *)
(* Rung L23 *)
IF (S103_M_차종1_AX OR S103_M_차종1_B OR S103_M_차종1_C OR S103_M_차종1_D OR S103_M_차종1_E OR S103_M_차종1_F OR S103_M_차종1_G OR S103_M_차종1_H) AND (S103_M_차종2_3DR OR S103_M_차종2_4DR OR S103_M_차종2_5DR OR S103_M_차종2_WGN OR S103_M_차종2_SP1 OR S103_M_차종2_SP2) AND (S103_M_차종3_LHD OR S103_M_차종3_RHD) AND (S103_M_차종4_내수 OR S103_M_차종4_수출 OR S103_M_차종4_북미 OR S103_M_차종4_EEC OR S103_M_차종4_호주 OR S103_M_차종4_중동 OR S103_M_차종4_중국 OR S103_M_차종4_브라질 OR S103_M_차종4_SP1 OR S103_M_차종4_SP2 OR S103_M_차종4_러시아 OR S103_M_차종4_SP3 OR S103_M_차종4_SP4 OR S103_M_차종4_SP5 OR S103_M_차종4_SP6 OR S103_M_차종4_SP7) AND (S103_M_차종5_MT OR S103_M_차종5_AT OR S103_M_차종5_SP1) AND (S103_M_차종6_일반루프 OR S103_M_차종6_썬루프 OR S103_M_차종6_파노라마루프 OR S103_M_차종6_DSROOF OR S103_M_차종6_SP1) AND (S103_M_차종7_GSL OR S103_M_차종7_DSL OR S103_M_차종7_SP1 OR S103_M_차종7_SP2 OR S103_M_차종7_SP3 OR S103_M_차종7_SP4 OR S103_M_차종7_SP5 OR S103_M_차종7_SP6) AND (S103_M_차종8_2WD OR S103_M_차종8_4WD OR S103_M_차종8_SP1) AND (S103_M_차종9_MPI OR S103_M_차종9_T_GDI OR S103_M_차종9_SP1 OR S103_M_차종9_SP2 OR S103_M_차종9_SP3 OR S103_M_차종9_SP4 OR S103_M_차종9_SP5 OR S103_M_차종9_SP6 OR S103_M_차종9_SP7 OR S103_M_차종9_SP8 OR S103_M_차종9_SP9 OR S103_M_차종9_SP10 OR S103_M_차종9_SP11) AND (S103_M_차종_OPT1_슬라이딩_유 OR S103_M_차종_OPT1_슬라이딩_무 OR S103_M_차종_OPT1_R_RACK_유 OR S103_M_차종_OPT1_R_RACK_무 OR S103_M_차종_OPT1_폴딩_유 OR S103_M_차종_OPT1_폴딩_무 OR S103_M_차종_OPT1_S_REP_EATER_유 OR S103_M_차종_OPT1_S_REP_EATER_무 OR S103_M_차종_OPT1_VAN_유 OR S103_M_차종_OPT1_VAN_무 OR S103_M_차종_OPT1_SP1 OR S103_M_차종_OPT1_SP2 OR S103_M_차종_OPT1_SP3 OR S103_M_차종_OPT1_SP4 OR S103_M_차종_OPT1_SP5 OR S103_M_차종_OPT1_SP6) THEN
    _t1 := S103_M_SEQ <> 0;
END_IF;
S103_M_STN_차종_ON := _t1;

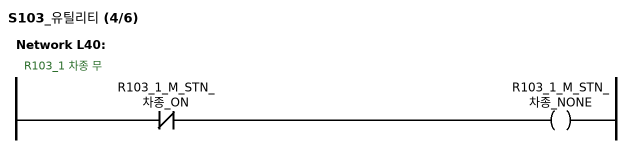
(* R103_1 차종 무 *)
(* Rung L40 *)
R103_1_M_STN_차종_NONE := NOT R103_1_M_STN_차종_ON;

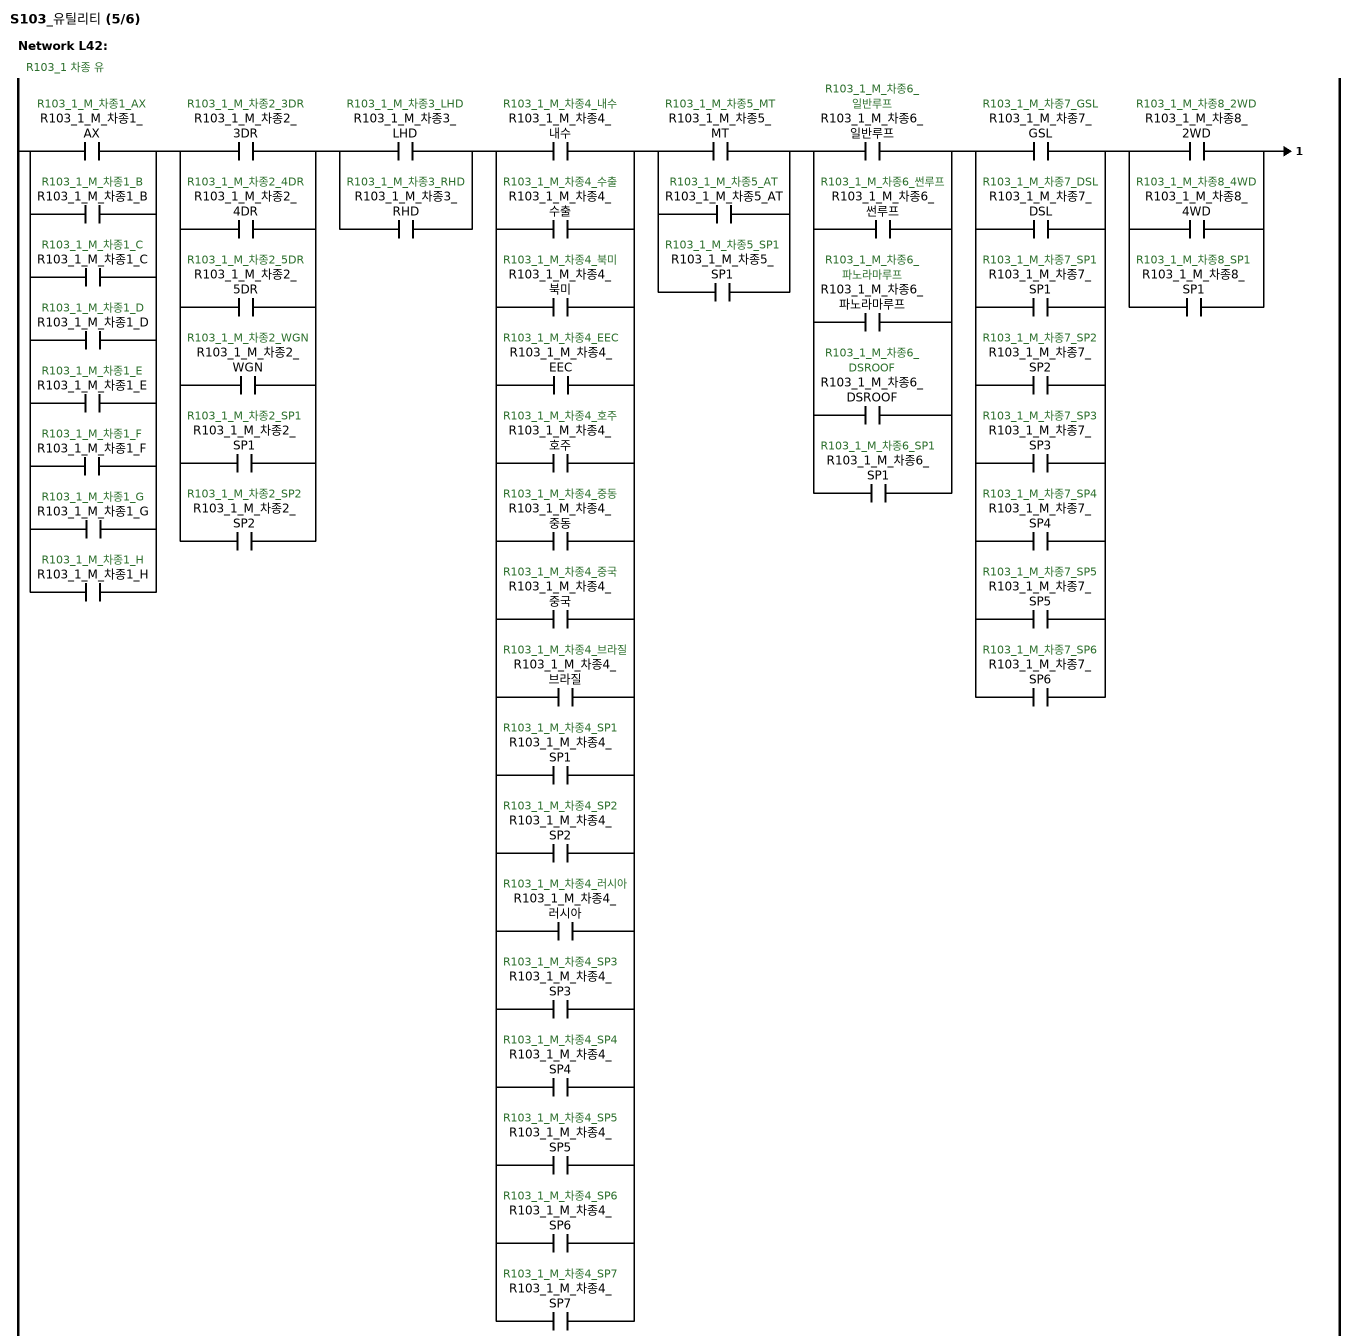

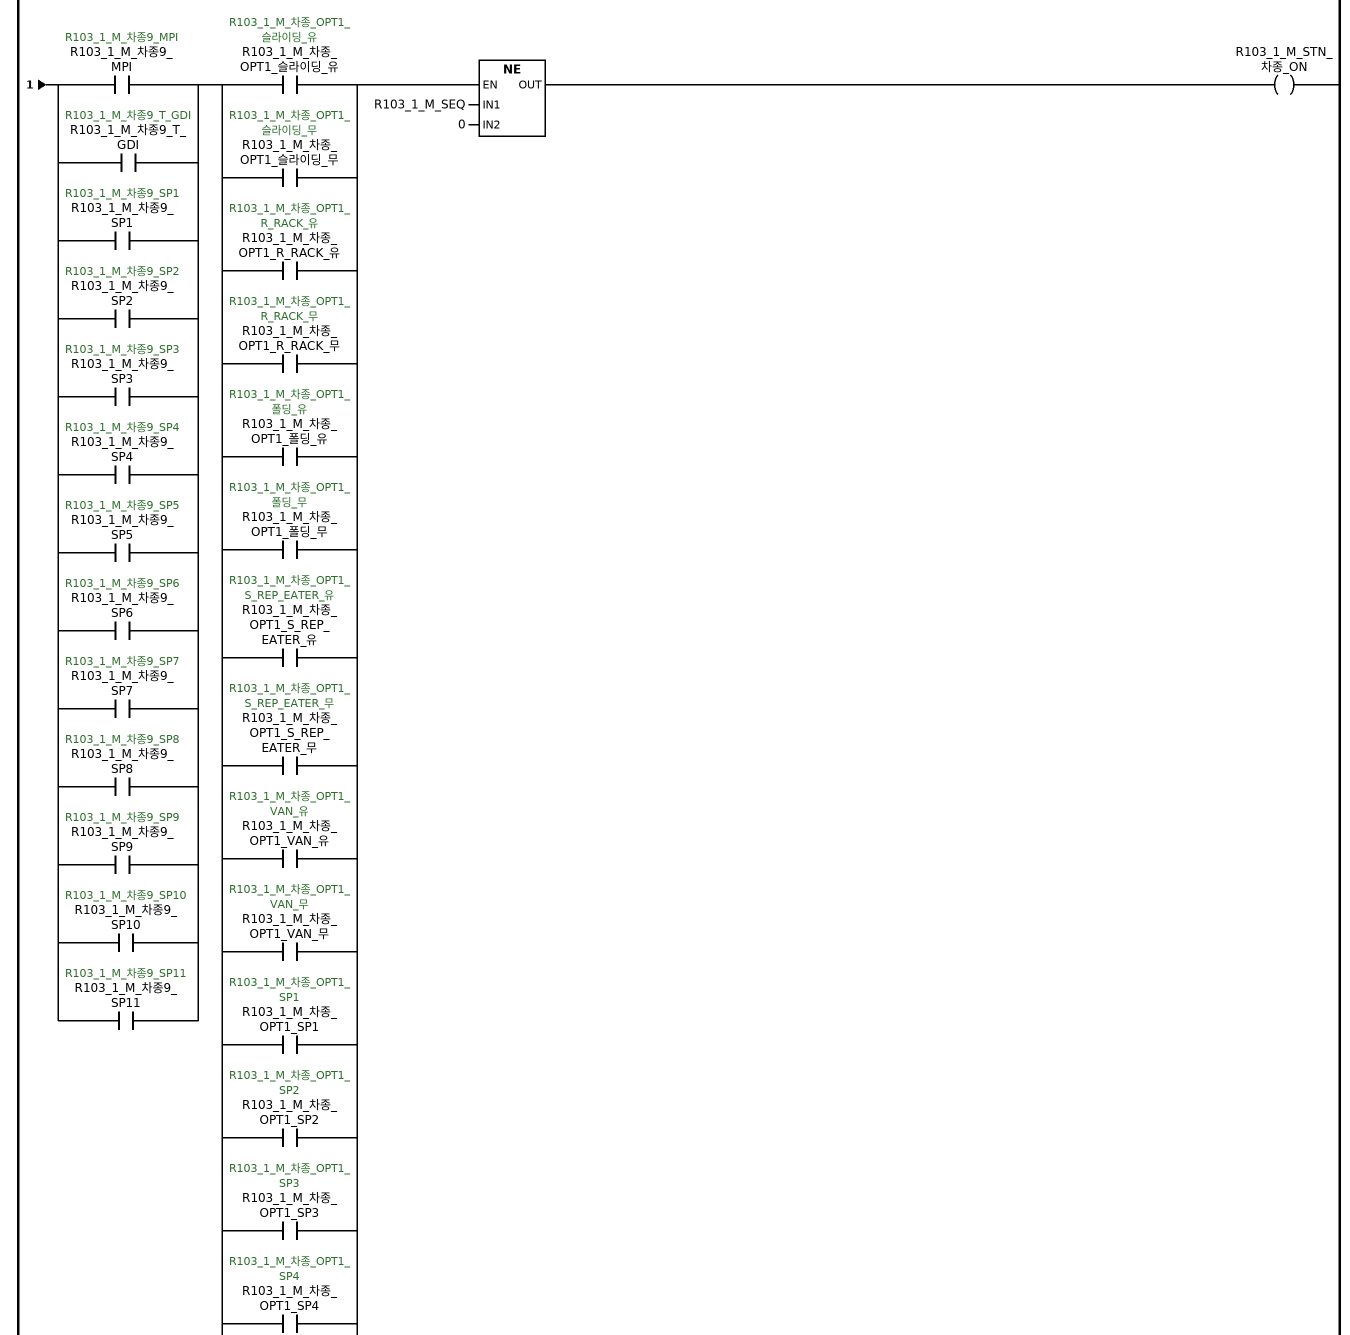

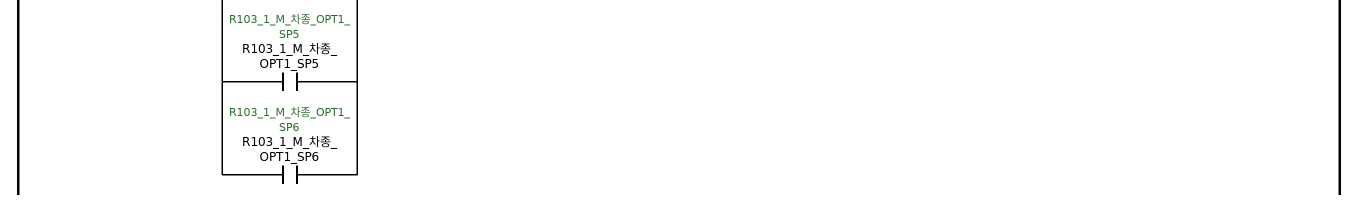
(* R103_1 차종 유 *)
(* Rung L42 *)
IF (R103_1_M_차종1_AX OR R103_1_M_차종1_B OR R103_1_M_차종1_C OR R103_1_M_차종1_D OR R103_1_M_차종1_E OR R103_1_M_차종1_F OR R103_1_M_차종1_G OR R103_1_M_차종1_H) AND (R103_1_M_차종2_3DR OR R103_1_M_차종2_4DR OR R103_1_M_차종2_5DR OR R103_1_M_차종2_WGN OR R103_1_M_차종2_SP1 OR R103_1_M_차종2_SP2) AND (R103_1_M_차종3_LHD OR R103_1_M_차종3_RHD) AND (R103_1_M_차종4_내수 OR R103_1_M_차종4_수출 OR R103_1_M_차종4_북미 OR R103_1_M_차종4_EEC OR R103_1_M_차종4_호주 OR R103_1_M_차종4_중동 OR R103_1_M_차종4_중국 OR R103_1_M_차종4_브라질 OR R103_1_M_차종4_SP1 OR R103_1_M_차종4_SP2 OR R103_1_M_차종4_러시아 OR R103_1_M_차종4_SP3 OR R103_1_M_차종4_SP4 OR R103_1_M_차종4_SP5 OR R103_1_M_차종4_SP6 OR R103_1_M_차종4_SP7) AND (R103_1_M_차종5_MT OR R103_1_M_차종5_AT OR R103_1_M_차종5_SP1) AND (R103_1_M_차종6_일반루프 OR R103_1_M_차종6_썬루프 OR R103_1_M_차종6_파노라마루프 OR R103_1_M_차종6_DSROOF OR R103_1_M_차종6_SP1) AND (R103_1_M_차종7_GSL OR R103_1_M_차종7_DSL OR R103_1_M_차종7_SP1 OR R103_1_M_차종7_SP2 OR R103_1_M_차종7_SP3 OR R103_1_M_차종7_SP4 OR R103_1_M_차종7_SP5 OR R103_1_M_차종7_SP6) AND (R103_1_M_차종8_2WD OR R103_1_M_차종8_4WD OR R103_1_M_차종8_SP1) AND (R103_1_M_차종9_MPI OR R103_1_M_차종9_T_GDI OR R103_1_M_차종9_SP1 OR R103_1_M_차종9_SP2 OR R103_1_M_차종9_SP3 OR R103_1_M_차종9_SP4 OR R103_1_M_차종9_SP5 OR R103_1_M_차종9_SP6 OR R103_1_M_차종9_SP7 OR R103_1_M_차종9_SP8 OR R103_1_M_차종9_SP9 OR R103_1_M_차종9_SP10 OR R103_1_M_차종9_SP11) AND (R103_1_M_차종_OPT1_슬라이딩_유 OR R103_1_M_차종_OPT1_슬라이딩_무 OR R103_1_M_차종_OPT1_R_RACK_유 OR R103_1_M_차종_OPT1_R_RACK_무 OR R103_1_M_차종_OPT1_폴딩_유 OR R103_1_M_차종_OPT1_폴딩_무 OR R103_1_M_차종_OPT1_S_REP_EATER_유 OR R103_1_M_차종_OPT1_S_REP_EATER_무 OR R103_1_M_차종_OPT1_VAN_유 OR R103_1_M_차종_OPT1_VAN_무 OR R103_1_M_차종_OPT1_SP1 OR R103_1_M_차종_OPT1_SP2 OR R103_1_M_차종_OPT1_SP3 OR R103_1_M_차종_OPT1_SP4 OR R103_1_M_차종_OPT1_SP5 OR R103_1_M_차종_OPT1_SP6) THEN
    _t2 := R103_1_M_SEQ <> 0;
END_IF;
R103_1_M_STN_차종_ON := _t2;

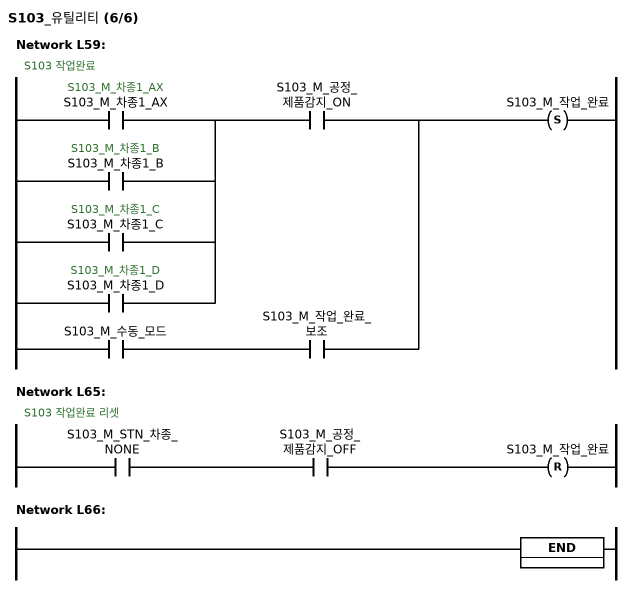
(* S103 작업완료 *)
(* Rung L59 *)
IF ((S103_M_차종1_AX OR S103_M_차종1_B OR S103_M_차종1_C OR S103_M_차종1_D) AND S103_M_공정_제품감지_ON) OR (S103_M_수동_모드 AND S103_M_작업_완료_보조) THEN
    S103_M_작업_완료 := TRUE;
END_IF;
(* S103 작업완료 리셋 *)
(* Rung L65 *)
IF S103_M_STN_차종_NONE AND S103_M_공정_제품감지_OFF THEN S103_M_작업_완료 := FALSE; END_IF;
(* Rung L66 *)
END();
END_PROGRAM

PROGRAM S103_동작 (* task: 스캔 프로그램 *)
VAR_EXTERNAL
    AWAYS_ON : BOOL; (* AT %MW3.1 *)
    EGIS_EJS : BOOL;
    MCP_PBL_101_자동_운전 : BOOL; (* AT %MW87630.4 *) (* 입력 접점 04 *)
    MCP_PBL_103_4_자동_운전 : BOOL; (* AT %MW87630.10 *) (* 입력 접점 10 *)
    MCP_PBL_운전준비_ON : BOOL; (* AT %MW87630.0 *) (* 입력 접점 00 *)
    MCP_SSP_101_수동_선택 : BOOL; (* AT %MW87630.2 *) (* 입력 접점 02 *)
    MCP_SSP_101_자동_선택 : BOOL; (* AT %MW87630.3 *) (* 입력 접점 03 *)
    MCP_SSP_103_4_수동_선택 : BOOL; (* AT %MW87630.8 *) (* 입력 접점 08 *)
    MCP_SSP_103_4_자동_선택 : BOOL; (* AT %MW87630.9 *) (* 입력 접점 09 *)
    S101_6_10_PLC_BOX_CP_TRIP : BOOL; (* AT %MW86102.15 *) (* 입력 접점 15 *)
    S101_AX_래치 : ACT_6_CYL;
    S101_HOME : BOOL; (* AT %MW1048.0 *)
    S101_M_ACT_선택_1 : BOOL; (* AT %MW1040.0 *)
    S101_M_ACT_선택_2 : BOOL; (* AT %MW1040.1 *)
    S101_M_AX_래치_전진_LAMP : WORD; (* AT %MW11100 *)
    S101_M_AX_래치_전진_LS_이상 : BOOL; (* AT %MW1100.5 *)
    S101_M_AX_래치_전진_보조 : BOOL; (* AT %MW1100.1 *)
    S101_M_AX_래치_전진단 : BOOL; (* AT %MW1100.3 *)
    S101_M_AX_래치_조건 : BOOL; (* AT %MW1100.0 *)
    S101_M_AX_래치_후진_LAMP : WORD; (* AT %MW11101 *)
    S101_M_AX_래치_후진_LS_이상 : BOOL; (* AT %MW1100.6 *)
    S101_M_AX_래치_후진_보조 : BOOL; (* AT %MW1100.2 *)
    S101_M_AX_래치_후진단 : BOOL; (* AT %MW1100.4 *)
    S101_M_SHIFT_전진_LAMP : WORD; (* AT %MW11102 *)
    S101_M_SHIFT_전진_LS_이상 : BOOL; (* AT %MW1101.5 *)
    S101_M_SHIFT_전진_보조 : BOOL; (* AT %MW1101.1 *)
    S101_M_SHIFT_전진단 : BOOL; (* AT %MW1101.3 *)
    S101_M_SHIFT_조건 : BOOL; (* AT %MW1101.0 *)
    S101_M_SHIFT_후진_LAMP : WORD; (* AT %MW11103 *)
    S101_M_SHIFT_후진_LS_이상 : BOOL; (* AT %MW1101.6 *)
    S101_M_SHIFT_후진_보조 : BOOL; (* AT %MW1101.2 *)
    S101_M_SHIFT_후진단 : BOOL; (* AT %MW1101.4 *)
    S101_M_STN_FRT_FLR_취출완료 : BOOL; (* AT %MW1001.13 *)
    S101_M_공정_APRON_제품감지_OFF : BOOL; (* AT %MW1001.4 *)
    S101_M_공정_APRON_제품감지_ON : BOOL; (* AT %MW1001.3 *)
    S101_M_공정_HOME_POSI : BOOL; (* AT %MW1004.0 *)
    S101_M_공정_간섭무 : BOOL; (* AT %MW1004.1 *)
    S101_M_수동_모드 : BOOL; (* AT %MW1000.3 *)
    S101_M_운전준비_ON : BOOL; (* AT %MW1000.0 *)
    S101_M_자동_START : BOOL; (* AT %MW1000.5 *)
    S101_M_자동_모드 : BOOL; (* AT %MW1000.1 *)
    S101_M_자동_운전중 : BOOL; (* AT %MW1000.4 *)
    S101_M_작업_완료 : BOOL; (* AT %MW1001.0 *)
    S101_M_총괄_CP_이상 : BOOL; (* AT %MW1009.7 *)
    S101_M_총괄_CT_이상 : BOOL; (* AT %MW1010.4 *)
    S101_M_총괄_EOCR_이상 : BOOL; (* AT %MW1009.8 *)
    S101_M_총괄_INV_이상 : BOOL; (* AT %MW1009.9 *)
    S101_M_총괄_LS_이상 : BOOL; (* AT %MW1009.15 *)
    S101_M_총괄_MATCH_이상 : BOOL; (* AT %MW1010.0 *)
    S101_M_총괄_MC_이상 : BOOL; (* AT %MW1009.13 *)
    S101_M_총괄_NFB_이상 : BOOL; (* AT %MW1009.11 *)
    S101_M_총괄_ROBOT_이상 : BOOL; (* AT %MW1010.1 *)
    S101_M_총괄_SAFETY_이상 : BOOL; (* AT %MW1009.2 *)
    S101_M_총괄_공기압_이상 : BOOL; (* AT %MW1009.3 *)
    S101_M_총괄_사양_이상 : BOOL; (* AT %MW1009.6 *)
    S101_M_총괄_오버런_이상 : BOOL; (* AT %MW1009.12 *)
    S101_M_총괄_용점타점수_이상 : BOOL; (* AT %MW1010.2 *)
    S101_M_총괄_이상 : BOOL; (* AT %MW1009.0 *)
    S101_M_총괄_제품감지_이상 : BOOL; (* AT %MW1009.4 *)
    S101_M_총괄_차종_이상 : BOOL; (* AT %MW1009.5 *)
    S101_M_총괄_통신_이상 : BOOL; (* AT %MW1009.14 *)
    S101_RS_AX_SFT_전진1 : BOOL; (* AT %MW86100.8 *) (* 입력 접점 08 *)
    S101_RS_AX_SFT_전진2 : BOOL; (* AT %MW86100.10 *) (* 입력 접점 10 *)
    S101_RS_AX_SFT_후진1 : BOOL; (* AT %MW86100.9 *) (* 입력 접점 09 *)
    S101_RS_AX_SFT_후진2 : BOOL; (* AT %MW86100.11 *) (* 입력 접점 11 *)
    S101_RS_AX_래치_전진1 : BOOL; (* AT %MW86100.0 *) (* 입력 접점 00 *)
    S101_RS_AX_래치_전진2 : BOOL; (* AT %MW86100.2 *) (* 입력 접점 02 *)
    S101_RS_AX_래치_후진1 : BOOL; (* AT %MW86100.1 *) (* 입력 접점 01 *)
    S101_RS_AX_래치_후진2 : BOOL; (* AT %MW86100.3 *) (* 입력 접점 03 *)
    S101_SHIFT : ACT_6_CYL;
    S101_SOL_AX_SHIFT_전진 : BOOL; (* AT %MW96103.2 *) (* 출력 접점 02 *)
    S101_SOL_AX_SHIFT_후진 : BOOL; (* AT %MW96103.3 *) (* 출력 접점 03 *)
    S101_SOL_AX_래치_전진 : BOOL; (* AT %MW96103.0 *) (* 출력 접점 00 *)
    S101_SOL_AX_래치_후진 : BOOL; (* AT %MW96103.1 *) (* 출력 접점 01 *)
    S101_전진_ON : BOOL; (* AT %MW1048.1 *)
    S101_후진_ON : BOOL; (* AT %MW1048.2 *)
    S102_M_차종1_AX : BOOL; (* AT %MW10061.0 *) (* S102_M_차종1_AX *)
    S103_6_30_PLC_BOX_CP_TRIP : BOOL; (* AT %MW86302.15 *) (* 입력 접점 15 *)
    S103_AX_래치 : ACT_6_CYL;
    S103_HOME : BOOL; (* AT %MW2048.0 *)
    S103_M_ACT_선택_1 : BOOL; (* AT %MW2040.0 *)
    S103_M_AX_래치_전진_LAMP : WORD; (* AT %MW12100 *)
    S103_M_AX_래치_전진_LS_이상 : BOOL; (* AT %MW2100.5 *)
    S103_M_AX_래치_전진_보조 : BOOL; (* AT %MW2100.1 *)
    S103_M_AX_래치_전진단 : BOOL; (* AT %MW2100.3 *)
    S103_M_AX_래치_조건 : BOOL; (* AT %MW2100.0 *)
    S103_M_AX_래치_후진_LAMP : WORD; (* AT %MW12101 *)
    S103_M_AX_래치_후진_LS_이상 : BOOL; (* AT %MW2100.6 *)
    S103_M_AX_래치_후진_보조 : BOOL; (* AT %MW2100.2 *)
    S103_M_AX_래치_후진단 : BOOL; (* AT %MW2100.4 *)
    S103_M_공정_HOME_POSI : BOOL; (* AT %MW2004.0 *)
    S103_M_공정_간섭무 : BOOL; (* AT %MW2004.1 *)
    S103_M_공정_제품감지_OFF : BOOL; (* AT %MW2001.4 *)
    S103_M_공정_제품감지_ON : BOOL; (* AT %MW2001.3 *)
    S103_M_수동_모드 : BOOL; (* AT %MW2000.3 *)
    S103_M_운전준비_ON : BOOL; (* AT %MW2000.0 *)
    S103_M_자동_START : BOOL; (* AT %MW2000.5 *)
    S103_M_자동_모드 : BOOL; (* AT %MW2000.1 *)
    S103_M_자동_운전중 : BOOL; (* AT %MW2000.4 *)
    S103_M_작업_완료 : BOOL; (* AT %MW2001.0 *)
    S103_M_총괄_CP_이상 : BOOL; (* AT %MW2009.7 *)
    S103_M_총괄_CT_이상 : BOOL; (* AT %MW2010.4 *)
    S103_M_총괄_EOCR_이상 : BOOL; (* AT %MW2009.8 *)
    S103_M_총괄_INV_이상 : BOOL; (* AT %MW2009.9 *)
    S103_M_총괄_LS_이상 : BOOL; (* AT %MW2009.15 *)
    S103_M_총괄_MATCH_이상 : BOOL; (* AT %MW2010.0 *)
    S103_M_총괄_MC_이상 : BOOL; (* AT %MW2009.13 *)
    S103_M_총괄_NFB_이상 : BOOL; (* AT %MW2009.11 *)
    S103_M_총괄_ROBOT_이상 : BOOL; (* AT %MW2010.1 *)
    S103_M_총괄_SAFETY_이상 : BOOL; (* AT %MW2009.2 *)
    S103_M_총괄_공기압_이상 : BOOL; (* AT %MW2009.3 *)
    S103_M_총괄_사양_이상 : BOOL; (* AT %MW2009.6 *)
    S103_M_총괄_오버런_이상 : BOOL; (* AT %MW2009.12 *)
    S103_M_총괄_용점타점수_이상 : BOOL; (* AT %MW2010.2 *)
    S103_M_총괄_이상 : BOOL; (* AT %MW2009.0 *)
    S103_M_총괄_제품감지_이상 : BOOL; (* AT %MW2009.4 *)
    S103_M_총괄_차종_이상 : BOOL; (* AT %MW2009.5 *)
    S103_M_총괄_통신_이상 : BOOL; (* AT %MW2009.14 *)
    S103_RS_AX_래치_전진1 : BOOL; (* AT %MW86300.0 *) (* 입력 접점 00 *)
    S103_RS_AX_래치_전진2 : BOOL; (* AT %MW86300.2 *) (* 입력 접점 02 *)
    S103_RS_AX_래치_전진3 : BOOL; (* AT %MW86300.4 *) (* 입력 접점 04 *)
    S103_RS_AX_래치_전진4 : BOOL; (* AT %MW86300.6 *) (* 입력 접점 06 *)
    S103_RS_AX_래치_후진1 : BOOL; (* AT %MW86300.1 *) (* 입력 접점 01 *)
    S103_RS_AX_래치_후진2 : BOOL; (* AT %MW86300.3 *) (* 입력 접점 03 *)
    S103_RS_AX_래치_후진3 : BOOL; (* AT %MW86300.5 *) (* 입력 접점 05 *)
    S103_RS_AX_래치_후진4 : BOOL; (* AT %MW86300.7 *) (* 입력 접점 07 *)
    S103_SOL_AX_래치_전진 : BOOL; (* AT %MW96303.0 *) (* 출력 접점 00 *)
    S103_SOL_AX_래치_후진 : BOOL; (* AT %MW96303.1 *) (* 출력 접점 01 *)
    S103_공기압_AIR_CHECK : BOOL; (* AT %MW86302.14 *) (* 입력 접점 14 *)
    S103_운전준비 : TON;
    S103_전진_ON : BOOL; (* AT %MW2048.1 *)
    S103_후진_ON : BOOL; (* AT %MW2048.2 *)
    T101_자동 : TON;
    T103_자동 : TON;
    전체_M_이상_리셋 : BOOL; (* AT %MW308.2 *) (* 전체 M 이상 리셋 *)
    전체_라인_M_총괄_SAFETY_이상 : BOOL; (* AT %MW300.2 *)
    전체_라인_M_총괄_공기압_이상 : BOOL; (* AT %MW300.3 *)
    전체_라인_M_총괄_비상정지_이상 : BOOL; (* AT %MW300.1 *)
    전체_라인_M_총괄_이상 : BOOL; (* AT %MW300.0 *)
END_VAR
VAR
    INST10 : TON;
    INST11 : TON;
    INST12 : TON;
    INST13 : TON;
    INST14 : TON;
    INST15 : TON;
    INST16 : TON;
    INST17 : TON;
    INST18 : TON;
    INST19 : TON;
    INST20 : TON;
    INST21 : TON;
    INST23 : TON;
    INST24 : TON;
    INST25 : TON;
    INST8 : TON;
    INST9 : TON;
END_VAR

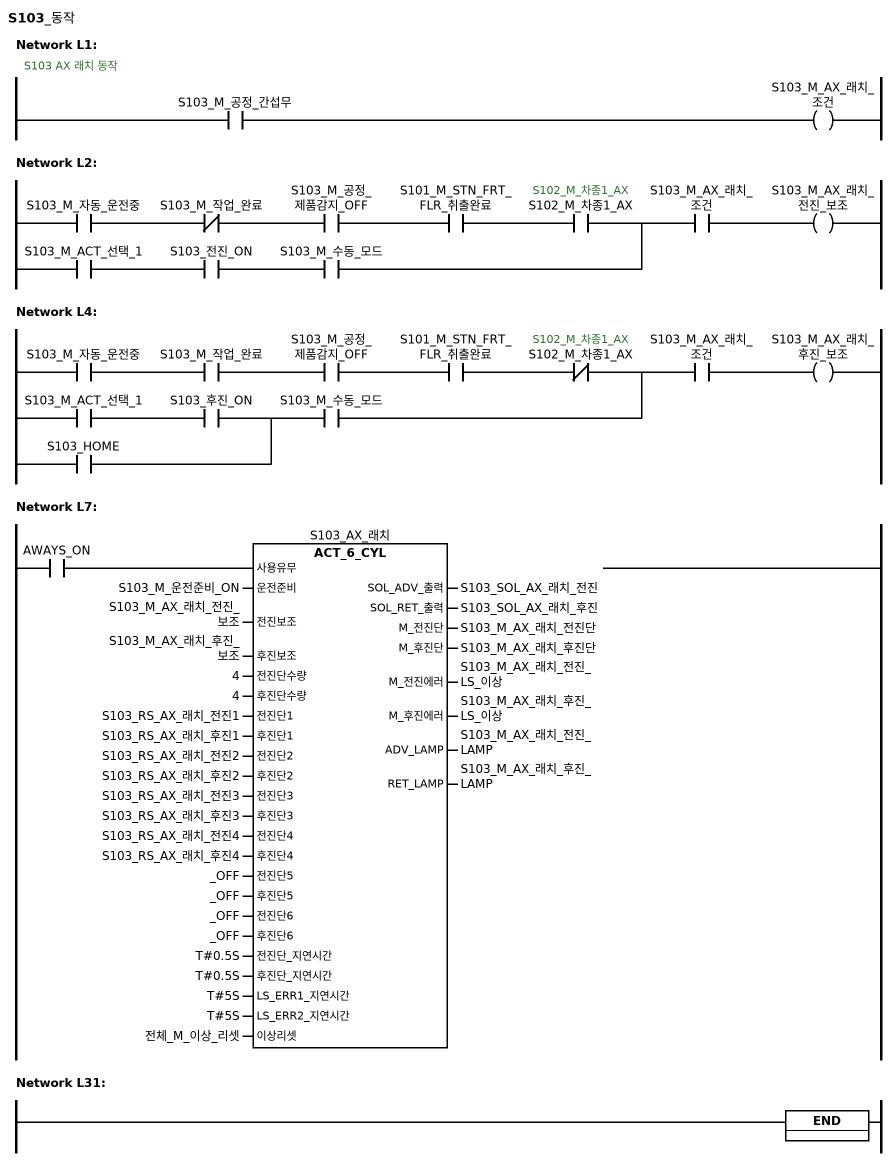
(* S103 AX 래치 동작 *)
(* Rung L1 *)
S103_M_AX_래치_조건 := S103_M_공정_간섭무;
(* Rung L2 *)
S103_M_AX_래치_전진_보조 := ((S103_M_자동_운전중 AND NOT S103_M_작업_완료 AND S103_M_공정_제품감지_OFF AND S101_M_STN_FRT_FLR_취출완료 AND S102_M_차종1_AX) OR (S103_M_ACT_선택_1 AND S103_전진_ON AND S103_M_수동_모드)) AND S103_M_AX_래치_조건;
(* Rung L4 *)
S103_M_AX_래치_후진_보조 := ((S103_M_자동_운전중 AND S103_M_작업_완료 AND S103_M_공정_제품감지_OFF AND S101_M_STN_FRT_FLR_취출완료 AND NOT S102_M_차종1_AX) OR (((S103_M_ACT_선택_1 AND S103_후진_ON) OR S103_HOME) AND S103_M_수동_모드)) AND S103_M_AX_래치_조건;
(* Rung L7 *)
S103_AX_래치(사용유무 := AWAYS_ON, 운전준비 := S103_M_운전준비_ON, 전진보조 := S103_M_AX_래치_전진_보조, 후진보조 := S103_M_AX_래치_후진_보조, 전진단수량 := 4, 후진단수량 := 4, 전진단1 := S103_RS_AX_래치_전진1, 후진단1 := S103_RS_AX_래치_후진1, 전진단2 := S103_RS_AX_래치_전진2, 후진단2 := S103_RS_AX_래치_후진2, 전진단3 := S103_RS_AX_래치_전진3, 후진단3 := S103_RS_AX_래치_후진3, 전진단4 := S103_RS_AX_래치_전진4, 후진단4 := S103_RS_AX_래치_후진4, 전진단5 := _OFF, 후진단5 := _OFF, 전진단6 := _OFF, 후진단6 := _OFF, 전진단_지연시간 := T#0.5S, 후진단_지연시간 := T#0.5S, LS_ERR1_지연시간 := T#5S, LS_ERR2_지연시간 := T#5S, 이상리셋 := 전체_M_이상_리셋, SOL_ADV_출력 => S103_SOL_AX_래치_전진, SOL_RET_출력 => S103_SOL_AX_래치_후진, M_전진단 => S103_M_AX_래치_전진단, M_후진단 => S103_M_AX_래치_후진단, M_전진에러 => S103_M_AX_래치_전진_LS_이상, M_후진에러 => S103_M_AX_래치_후진_LS_이상, ADV_LAMP => S103_M_AX_래치_전진_LAMP, RET_LAMP => S103_M_AX_래치_후진_LAMP);
(* Rung L31 *)
END();
END_PROGRAM

PROGRAM S103_로보트 (* task: 스캔 프로그램 *)
VAR_EXTERNAL
    AWAYS_OFF : BOOL; (* AT %MW3.0 *)
    AWAYS_ON : BOOL; (* AT %MW3.1 *)
    F_COMPL_I_불간섭 : BOOL; (* AT %MW83211.0 *)
    F_COMPL_I_자동_운전중 : BOOL; (* AT %MW83210.3 *)
    F_COMPL_I_진입OK : BOOL; (* AT %MW83211.1 *)
    F_COMPL_I_파트_NONE : BOOL; (* AT %MW83210.9 *)
    MCP_M_부저_정지 : BOOL; (* AT %MW350.5 *)
    MCP_M_비상정지 : BOOL; (* AT %MW350.7 *)
    MCP_PBL_운전준비_ON : BOOL; (* AT %MW87630.0 *) (* 입력 접점 00 *)
    R102_1_M_I_RB_간섭무_2 : BOOL; (* AT %MW20082.1 *)
    R103_1_I_RB_INPUT : ARRAY[0..3] OF WORD; (* AT %MW84100 *)
    R103_1_M_I_RB_1차_작업완료 : BOOL; (* AT %MW20101.2 *)
    R103_1_M_I_RB_2차_작업완료 : BOOL; (* AT %MW20101.3 *)
    R103_1_M_I_RB_3차_작업완료 : BOOL; (* AT %MW20101.4 *)
    R103_1_M_I_RB_4차_작업완료 : BOOL; (* AT %MW20101.5 *)
    R103_1_M_I_RB_5차_작업완료 : BOOL; (* AT %MW20101.6 *)
    R103_1_M_I_RB_6차_작업완료 : BOOL; (* AT %MW20101.7 *)
    R103_1_M_I_RB_7차_작업완료 : BOOL; (* AT %MW20101.8 *)
    R103_1_M_I_RB_PAUSE_보조 : BOOL; (* AT %MW20100.5 *)
    R103_1_M_I_RB_PLC_RUN_CHK_이상 : BOOL; (* AT %MW20100.7 *)
    R103_1_M_I_RB_간섭무_1 : BOOL; (* AT %MW20102.0 *)
    R103_1_M_I_RB_간섭무_10 : BOOL; (* AT %MW20102.9 *)
    R103_1_M_I_RB_간섭무_11 : BOOL; (* AT %MW20102.10 *)
    R103_1_M_I_RB_간섭무_12 : BOOL; (* AT %MW20102.11 *)
    R103_1_M_I_RB_간섭무_2 : BOOL; (* AT %MW20102.1 *)
    R103_1_M_I_RB_간섭무_3 : BOOL; (* AT %MW20102.2 *)
    R103_1_M_I_RB_간섭무_4 : BOOL; (* AT %MW20102.3 *)
    R103_1_M_I_RB_간섭무_5 : BOOL; (* AT %MW20102.4 *)
    R103_1_M_I_RB_간섭무_6 : BOOL; (* AT %MW20102.5 *)
    R103_1_M_I_RB_간섭무_7 : BOOL; (* AT %MW20102.6 *)
    R103_1_M_I_RB_간섭무_8 : BOOL; (* AT %MW20102.7 *)
    R103_1_M_I_RB_간섭무_9 : BOOL; (* AT %MW20102.8 *)
    R103_1_M_I_RB_비상정지 : BOOL; (* AT %MW20100.4 *)
    R103_1_M_I_RB_운전준비 : BOOL; (* AT %MW20100.0 *)
    R103_1_M_I_RB_원위치 : BOOL; (* AT %MW20100.3 *)
    R103_1_M_I_RB_이상 : BOOL; (* AT %MW20100.2 *)
    R103_1_M_I_RB_자동 : BOOL; (* AT %MW20100.1 *)
    R103_1_M_I_RB_최종작업완료 : BOOL; (* AT %MW20101.0 *)
    R103_1_M_I_RB_프로그램_이상 : BOOL; (* AT %MW20100.6 *)
    R103_1_M_O_RB_1_CYCLE_SET : BOOL; (* AT %MW21100.3 *)
    R103_1_M_O_RB_1차_작업완료_리셋 : BOOL; (* AT %MW21102.0 *)
    R103_1_M_O_RB_2차_작업완료_리셋 : BOOL; (* AT %MW21102.1 *)
    R103_1_M_O_RB_2차_진입OK : BOOL; (* AT %MW21101.8 *)
    R103_1_M_O_RB_3차_작업완료_리셋 : BOOL; (* AT %MW21102.2 *)
    R103_1_M_O_RB_3차_진입OK : BOOL; (* AT %MW21101.9 *)
    R103_1_M_O_RB_4차_작업완료_리셋 : BOOL; (* AT %MW21102.3 *)
    R103_1_M_O_RB_4차_진입OK : BOOL; (* AT %MW21101.10 *)
    R103_1_M_O_RB_5차_작업완료_리셋 : BOOL; (* AT %MW21102.4 *)
    R103_1_M_O_RB_5차_진입OK : BOOL; (* AT %MW21101.11 *)
    R103_1_M_O_RB_6차_작업완료_리셋 : BOOL; (* AT %MW21102.5 *)
    R103_1_M_O_RB_6차_진입OK : BOOL; (* AT %MW21101.12 *)
    R103_1_M_O_RB_7차_작업완료_리셋 : BOOL; (* AT %MW21102.6 *)
    R103_1_M_O_RB_7차_진입OK : BOOL; (* AT %MW21101.13 *)
    R103_1_M_O_RB_ATD_OK : BOOL; (* AT %MW21100.6 *)
    R103_1_M_O_RB_PLT_10_진입OK : BOOL; (* AT %MW21103.10 *)
    R103_1_M_O_RB_PLT_11_진입OK : BOOL; (* AT %MW21103.11 *)
    R103_1_M_O_RB_PLT_12_진입OK : BOOL; (* AT %MW21103.12 *)
    R103_1_M_O_RB_PLT_1_진입OK : BOOL; (* AT %MW21103.1 *)
    R103_1_M_O_RB_PLT_2_진입OK : BOOL; (* AT %MW21103.2 *)
    R103_1_M_O_RB_PLT_3_진입OK : BOOL; (* AT %MW21103.3 *)
    R103_1_M_O_RB_PLT_4_진입OK : BOOL; (* AT %MW21103.4 *)
    R103_1_M_O_RB_PLT_5_진입OK : BOOL; (* AT %MW21103.5 *)
    R103_1_M_O_RB_PLT_6_진입OK : BOOL; (* AT %MW21103.6 *)
    R103_1_M_O_RB_PLT_7_진입OK : BOOL; (* AT %MW21103.7 *)
    R103_1_M_O_RB_PLT_8_진입OK : BOOL; (* AT %MW21103.8 *)
    R103_1_M_O_RB_PLT_9_진입OK : BOOL; (* AT %MW21103.9 *)
    R103_1_M_O_RB_PLT_카운터리셋_보조 : BOOL; (* AT %MW21100.10 *)
    R103_1_M_O_RB_RESTART_OK : BOOL; (* AT %MW21100.2 *)
    R103_1_M_O_RB_START_OK : BOOL; (* AT %MW21100.0 *)
    R103_1_M_O_RB_TEST_MODE_5000회 : BOOL; (* AT %MW21100.12 *)
    R103_1_M_O_RB_TIP_교체_시작 : BOOL; (* AT %MW21100.7 *)
    R103_1_M_O_RB_TIP_교체_완료 : BOOL; (* AT %MW21100.8 *)
    R103_1_M_O_RB_VIP_MODE : BOOL; (* AT %MW21100.11 *)
    R103_1_M_O_RB_냉각수_차단_요청 : BOOL; (* AT %MW21100.9 *)
    R103_1_M_O_RB_진입OK_AX차종 : BOOL; (* AT %MW21101.0 *)
    R103_1_M_O_RB_진입OK_B차종 : BOOL; (* AT %MW21101.1 *)
    R103_1_M_O_RB_진입OK_C차종 : BOOL; (* AT %MW21101.2 *)
    R103_1_M_O_RB_진입OK_D차종 : BOOL; (* AT %MW21101.3 *)
    R103_1_M_O_RB_진입OK_E차종 : BOOL; (* AT %MW21101.4 *)
    R103_1_M_O_RB_진입OK_F차종 : BOOL; (* AT %MW21101.5 *)
    R103_1_M_O_RB_진입OK_G차종 : BOOL; (* AT %MW21101.6 *)
    R103_1_M_O_RB_진입OK_H차종 : BOOL; (* AT %MW21101.7 *)
    R103_1_M_O_RB_최종_작업완료_리셋 : BOOL; (* AT %MW21100.5 *)
    R103_1_M_O_RB_프로그램_OK : BOOL; (* AT %MW21100.1 *)
    R103_1_M_RB_PROG_NO : WORD; (* AT %MW20104 *)
    R103_1_O_RB_OUTPUT : ARRAY[0..3] OF WORD; (* AT %MW94100 *)
    S102_M_공정_제품감지_ON : BOOL; (* AT %MW1501.3 *)
    S103_M_FRT_취출OK_POS : BOOL; (* AT %MW2004.9 *)
    S103_M_STN_차종_ON : BOOL; (* AT %MW2002.0 *)
    S103_M_공정_제품감지_ON : BOOL; (* AT %MW2001.3 *)
    S103_M_자동_START : BOOL; (* AT %MW2000.5 *)
    S103_M_자동_운전중 : BOOL; (* AT %MW2000.4 *)
    S103_M_작업_완료 : BOOL; (* AT %MW2001.0 *)
    S103_M_차종1_AX : BOOL; (* AT %MW10101.0 *) (* S103_M_차종1_AX *)
    S103_M_총괄_이상 : BOOL; (* AT %MW2009.0 *)
    로보트제외 : BOOL;
    전체_M_GATE_CYCLE_정지 : BOOL; (* AT %MW308.0 *) (* 전체 M GATE CYCLE STOP *)
    전체_M_GATE_비상정지_정상 : BOOL; (* AT %MW308.4 *)
    전체_M_운전준비_보조 : BOOL; (* AT %MW308.5 *)
    전체_M_이상_리셋 : BOOL; (* AT %MW308.2 *) (* 전체 M 이상 리셋 *)
    전체_공정_M_총괄_비상정지_정상 : BOOL; (* AT %MW304.1 *) (* 전체 공정 M 총괄 비상정지 정상 *)
END_VAR
VAR
    INST1 : FB494_Robot_Hyundai_HMMI_v1;
END_VAR
(* ladder body could not be read *)
END_PROGRAM

PROGRAM S103_이상 (* task: 스캔 프로그램 *)
VAR
    INST10 : TON;
    INST11 : TON;
    INST12 : TON;
    INST13 : TON;
    INST14 : TON;
    INST15 : TON;
    INST16 : TON;
    INST17 : TON;
    INST18 : TON;
    INST19 : TON;
    INST20 : TON;
    INST21 : TON;
    INST22 : TON;
    INST23 : TON;
    INST24 : TON;
    INST25 : TON;
    INST8 : TON;
    INST9 : TON;
END_VAR
VAR_EXTERNAL
    R103_1_M_RB_통신이상 : BOOL; (* AT %MW2024.1 *)
    S102_M_총괄_비상정지_이상 : BOOL; (* AT %MW1509.1 *)
    S103_6_30_PLC_BOX_CP_TRIP : BOOL; (* AT %MW86302.15 *) (* 입력 접점 15 *)
    S103_M_AX_래치_전진_LS_이상 : BOOL; (* AT %MW2100.5 *)
    S103_M_AX_래치_후진_LS_이상 : BOOL; (* AT %MW2100.6 *)
    S103_M_STN_FRT_FLR_로딩완료 : BOOL; (* AT %MW2001.8 *)
    S103_M_공정_간섭무 : BOOL; (* AT %MW2004.1 *)
    S103_M_공정_통신이상 : BOOL; (* AT %MW2024.0 *)
    S103_M_제품감지_이상 : BOOL; (* AT %MW2014.0 *)
    S103_M_총괄_CP_이상 : BOOL; (* AT %MW2009.7 *)
    S103_M_총괄_CT_이상 : BOOL; (* AT %MW2010.4 *)
    S103_M_총괄_EOCR_이상 : BOOL; (* AT %MW2009.8 *)
    S103_M_총괄_INV_이상 : BOOL; (* AT %MW2009.9 *)
    S103_M_총괄_LS_이상 : BOOL; (* AT %MW2009.15 *)
    S103_M_총괄_MATCH_이상 : BOOL; (* AT %MW2010.0 *)
    S103_M_총괄_MC_이상 : BOOL; (* AT %MW2009.13 *)
    S103_M_총괄_NFB_이상 : BOOL; (* AT %MW2009.11 *)
    S103_M_총괄_ROBOT_이상 : BOOL; (* AT %MW2010.1 *)
    S103_M_총괄_SAFETY_이상 : BOOL; (* AT %MW2009.2 *)
    S103_M_총괄_공기압_이상 : BOOL; (* AT %MW2009.3 *)
    S103_M_총괄_비상정지_이상 : BOOL; (* AT %MW2009.1 *)
    S103_M_총괄_사양_이상 : BOOL; (* AT %MW2009.6 *)
    S103_M_총괄_오버런_이상 : BOOL; (* AT %MW2009.12 *)
    S103_M_총괄_용점타점수_이상 : BOOL; (* AT %MW2010.2 *)
    S103_M_총괄_이상 : BOOL; (* AT %MW2009.0 *)
    S103_M_총괄_제품감지_이상 : BOOL; (* AT %MW2009.4 *)
    S103_M_총괄_차종_이상 : BOOL; (* AT %MW2009.5 *)
    S103_M_총괄_통신_이상 : BOOL; (* AT %MW2009.14 *)
    S103_PRS_AX_제품감지_CHECK1 : BOOL; (* AT %MW86301.0 *) (* 입력 접점 00 *)
    S103_PRS_AX_제품감지_CHECK2 : BOOL; (* AT %MW86301.1 *) (* 입력 접점 01 *)
    S103_공기압_AIR_CHECK : BOOL; (* AT %MW86302.14 *) (* 입력 접점 14 *)
    _0004_EB10_CFG_ER : BOOL; (* AT %MX59640 *) (* EB 구성 에러 *)
    _0004_EB10_DEER : BOOL; (* AT %MX59641 *) (* EB 운전 중 탈락 *)
    _0006_EB10_CFG_ER : BOOL; (* AT %MW186022.0 *) (* EB 구성 에러 *)
    _0006_EB10_DEER : BOOL; (* AT %MW186022.1 *) (* EB 운전 중 탈락 *)
    _0006_EB10_IO_DEER : BOOL; (* AT %MW186023.2 *) (* EB IO 탈락 에러 *)
    _0006_EB10_IO_TYER : BOOL; (* AT %MW186023.1 *) (* EB IO 타입 에러 *)
    _0006_EB30_CFG_ER : BOOL; (* AT %MW186034.0 *) (* EB 구성 에러 *)
    _0006_EB30_DEER : BOOL; (* AT %MW186034.1 *) (* EB 운전 중 탈락 *)
    _0006_EB30_IO_DEER : BOOL; (* AT %MW186035.2 *) (* EB IO 탈락 에러 *)
    _0006_EB30_IO_TYER : BOOL; (* AT %MW186035.1 *) (* EB IO 타입 에러 *)
    전체_M_이상_리셋 : BOOL; (* AT %MW308.2 *) (* 전체 M 이상 리셋 *)
END_VAR

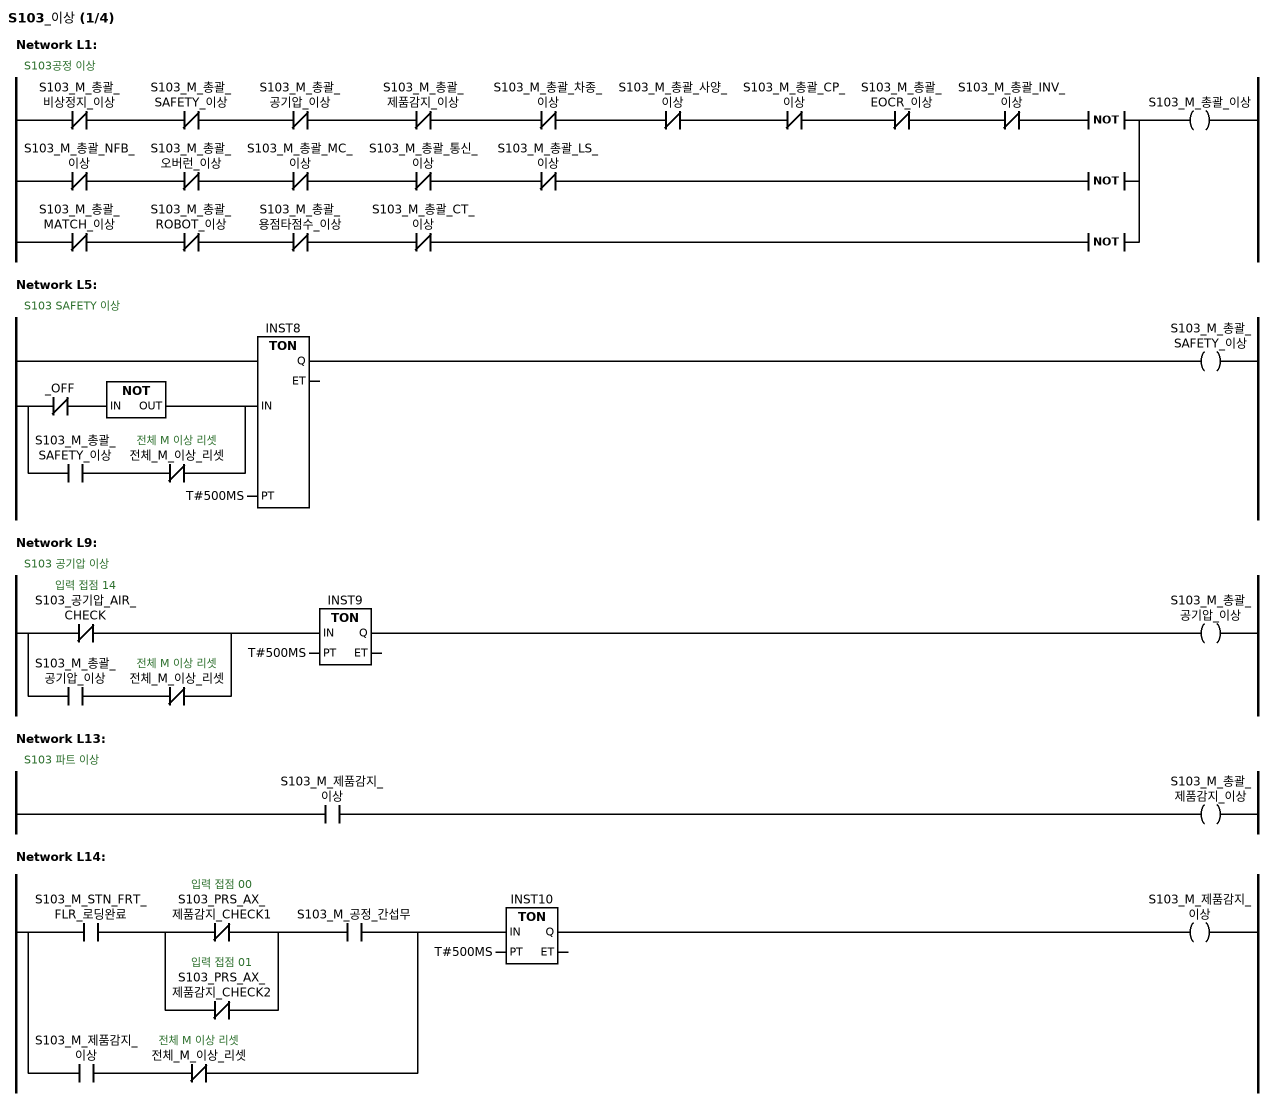
(* S103공정 이상 *)
(* Rung L1 *)
S103_M_총괄_이상 := NOT (NOT S103_M_총괄_비상정지_이상 AND NOT S103_M_총괄_SAFETY_이상 AND NOT S103_M_총괄_공기압_이상 AND NOT S103_M_총괄_제품감지_이상 AND NOT S103_M_총괄_차종_이상 AND NOT S103_M_총괄_사양_이상 AND NOT S103_M_총괄_CP_이상 AND NOT S103_M_총괄_EOCR_이상 AND NOT S103_M_총괄_INV_이상) OR NOT (NOT S103_M_총괄_NFB_이상 AND NOT S103_M_총괄_오버런_이상 AND NOT S103_M_총괄_MC_이상 AND NOT S103_M_총괄_통신_이상 AND NOT S103_M_총괄_LS_이상) OR NOT (NOT S103_M_총괄_MATCH_이상 AND NOT S103_M_총괄_ROBOT_이상 AND NOT S103_M_총괄_용점타점수_이상 AND NOT S103_M_총괄_CT_이상);
(* S103 SAFETY 이상 *)
(* Rung L5 *)
INST8(IN := (NOT (NOT _OFF)) OR (S103_M_총괄_SAFETY_이상 AND NOT 전체_M_이상_리셋), PT := T#500MS);
S103_M_총괄_SAFETY_이상 := INST8.Q;
(* S103 공기압 이상 *)
(* Rung L9 *)
INST9(IN := NOT S103_공기압_AIR_CHECK OR (S103_M_총괄_공기압_이상 AND NOT 전체_M_이상_리셋), PT := T#500MS);
S103_M_총괄_공기압_이상 := INST9.Q;
(* S103 파트 이상 *)
(* Rung L13 *)
S103_M_총괄_제품감지_이상 := S103_M_제품감지_이상;
(* Rung L14 *)
INST10(IN := (S103_M_STN_FRT_FLR_로딩완료 AND (NOT S103_PRS_AX_제품감지_CHECK1 OR NOT S103_PRS_AX_제품감지_CHECK2) AND S103_M_공정_간섭무) OR (S103_M_제품감지_이상 AND NOT 전체_M_이상_리셋), PT := T#500MS);
S103_M_제품감지_이상 := INST10.Q;

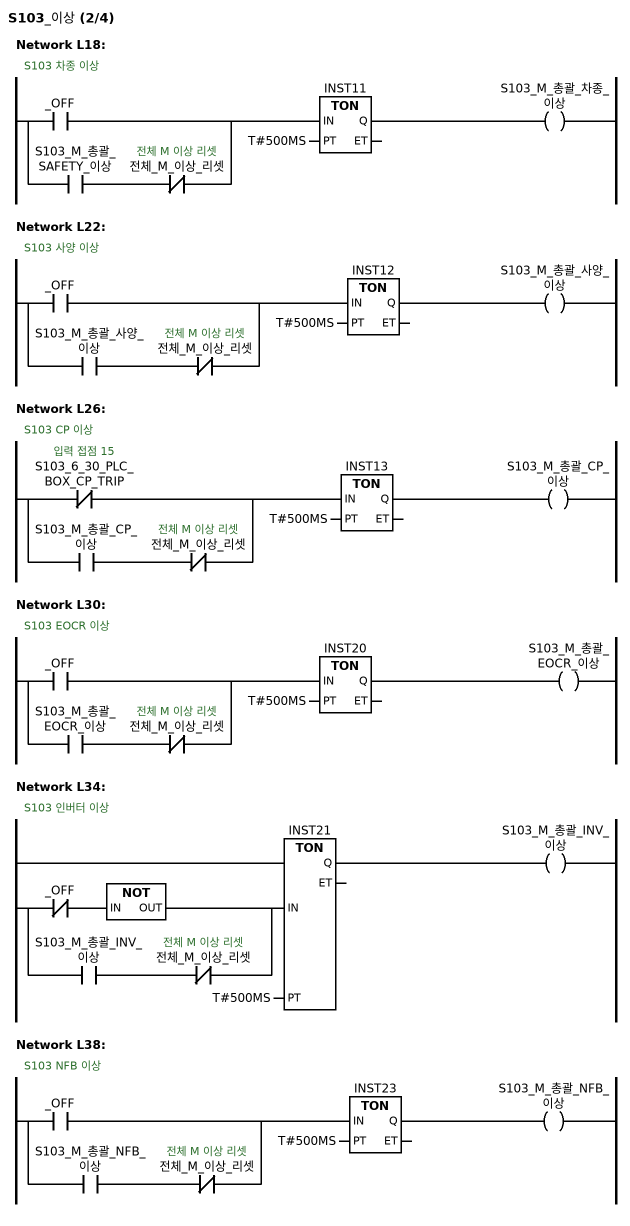
(* S103 차종 이상 *)
(* Rung L18 *)
INST11(IN := _OFF OR (S103_M_총괄_SAFETY_이상 AND NOT 전체_M_이상_리셋), PT := T#500MS);
S103_M_총괄_차종_이상 := INST11.Q;
(* S103 사양 이상 *)
(* Rung L22 *)
INST12(IN := _OFF OR (S103_M_총괄_사양_이상 AND NOT 전체_M_이상_리셋), PT := T#500MS);
S103_M_총괄_사양_이상 := INST12.Q;
(* S103 CP 이상 *)
(* Rung L26 *)
INST13(IN := NOT S103_6_30_PLC_BOX_CP_TRIP OR (S103_M_총괄_CP_이상 AND NOT 전체_M_이상_리셋), PT := T#500MS);
S103_M_총괄_CP_이상 := INST13.Q;
(* S103 EOCR 이상 *)
(* Rung L30 *)
INST20(IN := _OFF OR (S103_M_총괄_EOCR_이상 AND NOT 전체_M_이상_리셋), PT := T#500MS);
S103_M_총괄_EOCR_이상 := INST20.Q;
(* S103 인버터 이상 *)
(* Rung L34 *)
INST21(IN := (NOT (NOT _OFF)) OR (S103_M_총괄_INV_이상 AND NOT 전체_M_이상_리셋), PT := T#500MS);
S103_M_총괄_INV_이상 := INST21.Q;
(* S103 NFB 이상 *)
(* Rung L38 *)
INST23(IN := _OFF OR (S103_M_총괄_NFB_이상 AND NOT 전체_M_이상_리셋), PT := T#500MS);
S103_M_총괄_NFB_이상 := INST23.Q;

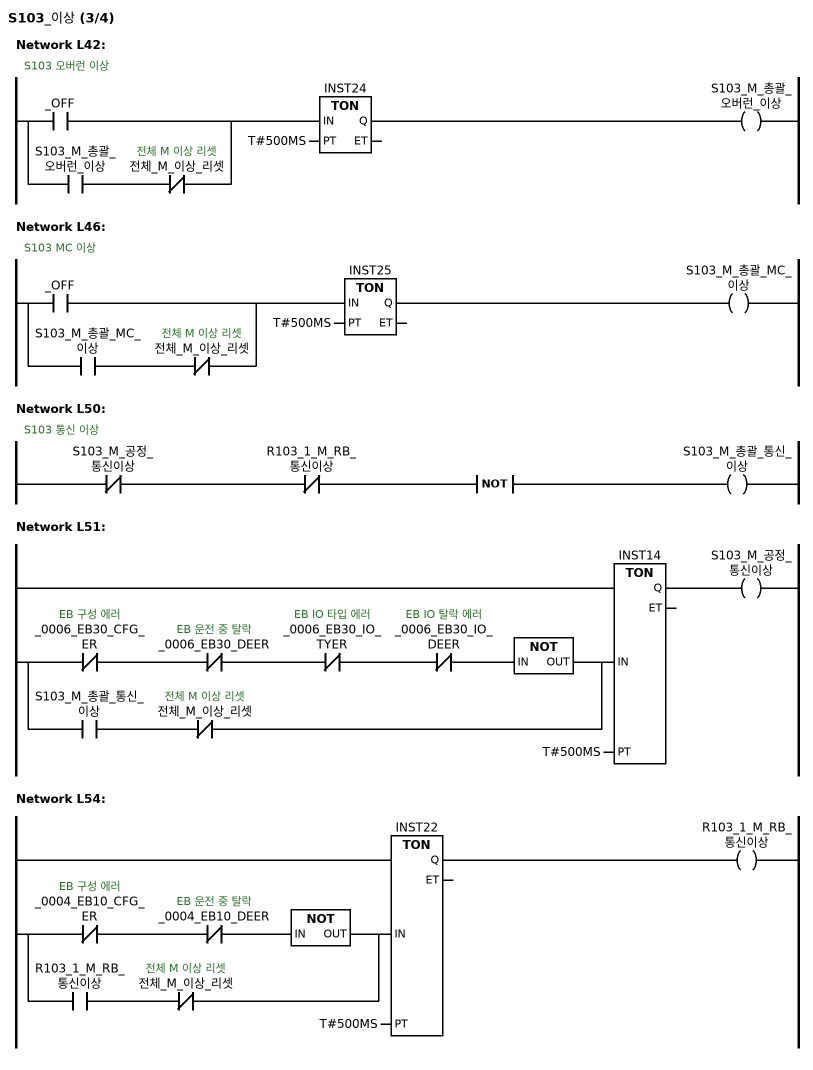
(* S103 오버런 이상 *)
(* Rung L42 *)
INST24(IN := _OFF OR (S103_M_총괄_오버런_이상 AND NOT 전체_M_이상_리셋), PT := T#500MS);
S103_M_총괄_오버런_이상 := INST24.Q;
(* S103 MC 이상 *)
(* Rung L46 *)
INST25(IN := _OFF OR (S103_M_총괄_MC_이상 AND NOT 전체_M_이상_리셋), PT := T#500MS);
S103_M_총괄_MC_이상 := INST25.Q;
(* S103 통신 이상 *)
(* Rung L50 *)
S103_M_총괄_통신_이상 := NOT (NOT S103_M_공정_통신이상 AND NOT R103_1_M_RB_통신이상);
(* Rung L51 *)
INST14(IN := (NOT (NOT _0006_EB30_CFG_ER AND NOT _0006_EB30_DEER AND NOT _0006_EB30_IO_TYER AND NOT _0006_EB30_IO_DEER)) OR (S103_M_총괄_통신_이상 AND NOT 전체_M_이상_리셋), PT := T#500MS);
S103_M_공정_통신이상 := INST14.Q;
(* Rung L54 *)
INST22(IN := (NOT (NOT _0004_EB10_CFG_ER AND NOT _0004_EB10_DEER)) OR (R103_1_M_RB_통신이상 AND NOT 전체_M_이상_리셋), PT := T#500MS);
R103_1_M_RB_통신이상 := INST22.Q;

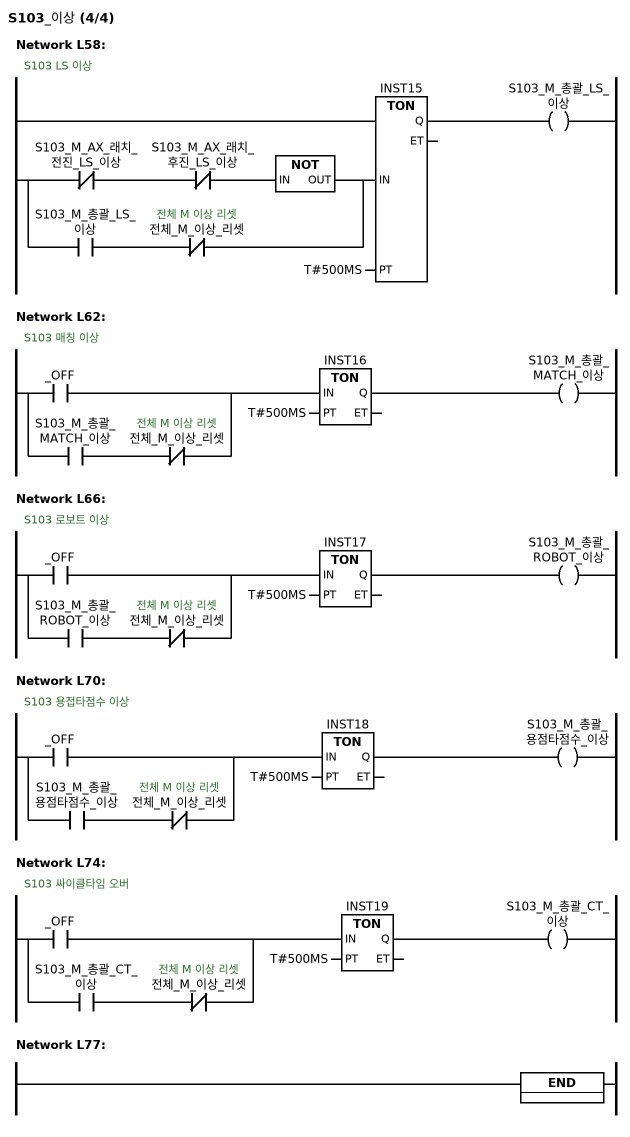
(* S103 LS 이상 *)
(* Rung L58 *)
INST15(IN := (NOT (NOT S103_M_AX_래치_전진_LS_이상 AND NOT S103_M_AX_래치_후진_LS_이상)) OR (S103_M_총괄_LS_이상 AND NOT 전체_M_이상_리셋), PT := T#500MS);
S103_M_총괄_LS_이상 := INST15.Q;
(* S103 매칭 이상 *)
(* Rung L62 *)
INST16(IN := _OFF OR (S103_M_총괄_MATCH_이상 AND NOT 전체_M_이상_리셋), PT := T#500MS);
S103_M_총괄_MATCH_이상 := INST16.Q;
(* S103 로보트 이상 *)
(* Rung L66 *)
INST17(IN := _OFF OR (S103_M_총괄_ROBOT_이상 AND NOT 전체_M_이상_리셋), PT := T#500MS);
S103_M_총괄_ROBOT_이상 := INST17.Q;
(* S103 용접타점수 이상 *)
(* Rung L70 *)
INST18(IN := _OFF OR (S103_M_총괄_용점타점수_이상 AND NOT 전체_M_이상_리셋), PT := T#500MS);
S103_M_총괄_용점타점수_이상 := INST18.Q;
(* S103 싸이클타임 오버 *)
(* Rung L74 *)
INST19(IN := _OFF OR (S103_M_총괄_CT_이상 AND NOT 전체_M_이상_리셋), PT := T#500MS);
S103_M_총괄_CT_이상 := INST19.Q;
(* Rung L77 *)
END();
END_PROGRAM

PROGRAM F_COMPL_라인인터록 (* task: 스캔 프로그램 *)
VAR_EXTERNAL
    AWAYS_OFF : BOOL; (* AT %MW3.0 *)
    CLOCK_BIT_0_5Sec : BOOL; (* AT %MW0.3 *)
    F_COMPL_I_차종수신완료 : BOOL; (* AT %MW83211.4 *)
    F_COMPL_I_차종요구 : BOOL; (* AT %MW83211.3 *)
    F_COMPL_O_SAFTY_이상 : BOOL; (* AT %MW93210.14 *)
    F_COMPL_O_불간섭 : BOOL; (* AT %MW93211.0 *)
    F_COMPL_O_비상정지 : BOOL; (* AT %MW93210.15 *)
    F_COMPL_O_수동모드 : BOOL; (* AT %MW93210.1 *)
    F_COMPL_O_운전준비 : BOOL; (* AT %MW93210.0 *)
    F_COMPL_O_자동_운전중 : BOOL; (* AT %MW93210.3 *)
    F_COMPL_O_자동모드 : BOOL; (* AT %MW93210.2 *)
    F_COMPL_O_작업완료 : BOOL; (* AT %MW93211.5 *)
    F_COMPL_O_총괄_이상 : BOOL; (* AT %MW93210.13 *)
    F_COMPL_O_통신_CHK : BOOL; (* AT %MW93211.15 *)
    R103_1_M_I_RB_간섭무_2 : BOOL; (* AT %MW20102.1 *)
    R103_1_M_I_RB_운전준비 : BOOL; (* AT %MW20100.0 *)
    R103_1_M_I_RB_이상 : BOOL; (* AT %MW20100.2 *)
    R103_1_M_I_RB_최종작업완료 : BOOL; (* AT %MW20101.0 *)
    R103_1_M_SEQ : WORD; (* AT %MW10120 *) (* R103_1_M_SEQ *)
    S103_M_수동_모드 : BOOL; (* AT %MW2000.3 *)
    S103_M_운전준비_ON : BOOL; (* AT %MW2000.0 *)
    S103_M_자동_START : BOOL; (* AT %MW2000.5 *)
    S103_M_자동_모드 : BOOL; (* AT %MW2000.1 *)
    S103_M_총괄_이상 : BOOL; (* AT %MW2009.0 *)
    전체_라인_M_총괄_비상정지_이상 : BOOL; (* AT %MW300.1 *)
END_VAR

